LIN {X 0,Y 394.469,Z 685.03,A -85,B 0,C 180,E1 10622.196,E2 10622.196} C_VEL
LIN {X 0,Y 393.966,Z 685.03,A -85,B 0,C 180,E1 10628.817,E2 10628.817} C_VEL
LIN {X 0,Y 393.674,Z 685.03,A -85,B 0,C 180,E1 10635.567,E2 10635.567} C_VEL
LIN {X 0,Y 393.333,Z 685.03,A -85,B 0,C 180,E1 10642.965,E2 10642.965} C_VEL
LIN {X 0,Y 393.105,Z 685.03,A -85,B 0,C 180,E1 10649.938,E2 10649.938} C_VEL
LIN {X 0,Y 392.893,Z 685.03,A -85,B 0,C 180,E1 10656.24,E2 10656.24} C_VEL
LIN {X 0,Y 392.936,Z 685.03,A -85,B 0,C 180,E1 10662.119,E2 10662.119} C_VEL
LIN {X 0,Y 395.462,Z 690.771,A -85,B 0,C 180,E1 10662.638,E2 10662.638} C_VEL
LIN {X 0,Y 416.78,Z 729.542,A -85,B 0,C 180,E1 10666.332,E2 10666.332} C_VEL
LIN {X 0,Y 428.209,Z 756.474,A -85,B 0,C 180,E1 10668.361,E2 10668.361} C_VEL
LIN {X 0,Y 424.245,Z 796.711,A -85,B 0,C 180,E1 10669.819,E2 10669.819} C_VEL
LIN {X 0,Y 419.16,Z 833.859,A -85,B 0,C 180,E1 10671.939,E2 10671.939} C_VEL
LIN {X 0,Y 413.098,Z 871.588,A -85,B 0,C 180,E1 10675.018,E2 10675.018} C_VEL
LIN {X 0,Y 407.027,Z 907.214,A -85,B 0,C 180,E1 10679.043,E2 10679.043} C_VEL
LIN {X 0,Y 402.042,Z 937.236,A -85,B 0,C 180,E1 10683.592,E2 10683.592} C_VEL
LIN {X 0,Y 398.385,Z 962.296,A -85,B 0,C 180,E1 10688.625,E2 10688.625} C_VEL
LIN {X 0,Y 396.268,Z 980.981,A -85,B 0,C 180,E1 10693.688,E2 10693.688} C_VEL
LIN {X 0,Y 395.371,Z 993.17,A -85,B 0,C 180,E1 10698.288,E2 10698.288} C_VEL
LIN {X 0,Y 392.685,Z 996.516,A -85,B 0,C 180,E1 10700.091,E2 10700.091} C_VEL
LIN {X 0,Y 387.255,Z 999.958,A -85,B 0,C 180,E1 10702.863,E2 10702.863} C_VEL
LIN {X 0,Y 387.166,Z 1000.335,A -85,B 0,C 180,E1 10703.185,E2 10703.185} C_VEL
LIN {X 0,Y 387.072,Z 1004.062,A -85,B 0,C 180,E1 10707.766,E2 10707.766} C_VEL
LIN {X 0,Y 387.105,Z 1004.068,A -85,B 0,C 180,E1 10712.234,E2 10712.234} C_VEL
LIN {X 0,Y 387.212,Z 999.067,A -85,B 0,C 180,E1 10717.839,E2 10717.839} C_VEL
LIN {X 0,Y 387.791,Z 988.198,A -85,B 0,C 180,E1 10723.502,E2 10723.502} C_VEL
LIN {X 0,Y 389.429,Z 970.858,A -85,B 0,C 180,E1 10729.23,E2 10729.23} C_VEL
LIN {X 0,Y 392.649,Z 947.513,A -85,B 0,C 180,E1 10734.704,E2 10734.704} C_VEL
LIN {X 0,Y 397.331,Z 919.555,A -85,B 0,C 180,E1 10739.585,E2 10739.585} C_VEL
LIN {X 0,Y 403.125,Z 887.2,A -85,B 0,C 180,E1 10743.835,E2 10743.835} C_VEL
LIN {X 0,Y 409.473,Z 851.855,A -85,B 0,C 180,E1 10747.269,E2 10747.269} C_VEL
LIN {X 0,Y 415.531,Z 813.064,A -85,B 0,C 180,E1 10749.969,E2 10749.969} C_VEL
LIN {X 0,Y 420.802,Z 771.94,A -85,B 0,C 180,E1 10751.807,E2 10751.807} C_VEL
LIN {X 0,Y 421.503,Z 758.027,A -85,B 0,C 180,E1 10752.3,E2 10752.3} C_VEL
LIN {X 0,Y 406.47,Z 724.052,A -85,B 0,C 180,E1 10755.061,E2 10755.061} C_VEL
LIN {X 0,Y 386.866,Z 689.928,A -85,B 0,C 180,E1 10758.649,E2 10758.649} C_VEL
LIN {X 0,Y 385.156,Z 685.03,A -85,B 0,C 180,E1 10759.111,E2 10759.111} C_VEL
LIN {X 0,Y 385.205,Z 685.03,A -85,B 0,C 180,E1 10765.351,E2 10765.351} C_VEL
LIN {X 0,Y 385.298,Z 685.03,A -85,B 0,C 180,E1 10771.965,E2 10771.965} C_VEL
LIN {X 0,Y 385.532,Z 685.03,A -85,B 0,C 180,E1 10779.371,E2 10779.371} C_VEL
LIN {X 0,Y 385.875,Z 685.03,A -85,B 0,C 180,E1 10786.427,E2 10786.427} C_VEL
LIN {X 0,Y 386.183,Z 685.03,A -85,B 0,C 180,E1 10793.264,E2 10793.264} C_VEL
LIN {X 0,Y 386.519,Z 685.03,A -85,B 0,C 180,E1 10799.996,E2 10799.996} C_VEL
LIN {X 0,Y 386.212,Z 685.03,A -85,B 0,C 180,E1 10806.727,E2 10806.727} C_VEL
LIN {X 0,Y 385.892,Z 685.03,A -85,B 0,C 180,E1 10813.564,E2 10813.564} C_VEL
LIN {X 0,Y 385.559,Z 685.03,A -85,B 0,C 180,E1 10820.618,E2 10820.618} C_VEL
LIN {X 0,Y 385.238,Z 685.03,A -85,B 0,C 180,E1 10828.03,E2 10828.03} C_VEL
LIN {X 0,Y 385.121,Z 685.03,A -85,B 0,C 180,E1 10835.988,E2 10835.988} C_VEL
LIN {X 0,Y 385.051,Z 685.03,A -85,B 0,C 180,E1 10841.875,E2 10841.875} C_VEL
LIN {X 0,Y 385.093,Z 685.261,A -85,B 0,C 180,E1 10847.204,E2 10847.204} C_VEL
LIN {X 0,Y 389.899,Z 695.532,A -85,B 0,C 180,E1 10848.478,E2 10848.478} C_VEL
LIN {X 0,Y 403.522,Z 724.973,A -85,B 0,C 180,E1 10852.426,E2 10852.426} C_VEL
LIN {X 0,Y 413.149,Z 753.666,A -85,B 0,C 180,E1 10856.345,E2 10856.345} C_VEL
LIN {X 0,Y 411.811,Z 765.062,A -85,B 0,C 180,E1 10857.501,E2 10857.501} C_VEL
LIN {X 0,Y 405.854,Z 793.487,A -85,B 0,C 180,E1 10860.821,E2 10860.821} C_VEL
LIN {X 0,Y 399.764,Z 819.011,A -85,B 0,C 180,E1 10864.93,E2 10864.93} C_VEL
LIN {X 0,Y 394.494,Z 840.743,A -85,B 0,C 180,E1 10869.863,E2 10869.863} C_VEL
LIN {X 0,Y 390.94,Z 856.405,A -85,B 0,C 180,E1 10875.016,E2 10875.016} C_VEL
LIN {X 0,Y 389.057,Z 866.332,A -85,B 0,C 180,E1 10879.948,E2 10879.948} C_VEL
LIN {X 0,Y 388.111,Z 872.539,A -85,B 0,C 180,E1 10885.54,E2 10885.54} C_VEL
LIN {X 0,Y 387.923,Z 874.065,A -85,B 0,C 180,E1 10890,E2 10890} C_VEL
LIN {X 0,Y 388.096,Z 872.475,A -85,B 0,C 180,E1 10894.46,E2 10894.46} C_VEL
LIN {X 0,Y 389.066,Z 866.191,A -85,B 0,C 180,E1 10900.051,E2 10900.051} C_VEL
LIN {X 0,Y 391.325,Z 854.489,A -85,B 0,C 180,E1 10905.66,E2 10905.66} C_VEL
LIN {X 0,Y 395.094,Z 837.935,A -85,B 0,C 180,E1 10910.788,E2 10910.788} C_VEL
LIN {X 0,Y 400.386,Z 816.384,A -85,B 0,C 180,E1 10915.461,E2 10915.461} C_VEL
LIN {X 0,Y 406.767,Z 789.56,A -85,B 0,C 180,E1 10919.616,E2 10919.616} C_VEL
LIN {X 0,Y 413.018,Z 758.951,A -85,B 0,C 180,E1 10922.981,E2 10922.981} C_VEL
LIN {X 0,Y 412.872,Z 752.781,A -85,B 0,C 180,E1 10923.689,E2 10923.689} C_VEL
LIN {X 0,Y 402.515,Z 722.507,A -85,B 0,C 180,E1 10927.806,E2 10927.806} C_VEL
LIN {X 0,Y 388.97,Z 693.749,A -85,B 0,C 180,E1 10931.663,E2 10931.663} C_VEL
LIN {X 0,Y 385.136,Z 685.03,A -85,B 0,C 180,E1 10932.792,E2 10932.792} C_VEL
LIN {X 0,Y 385.061,Z 685.03,A -85,B 0,C 180,E1 10938.235,E2 10938.235} C_VEL
LIN {X 0,Y 385.145,Z 685.03,A -85,B 0,C 180,E1 10944.015,E2 10944.015} C_VEL
LIN {X 0,Y 385.28,Z 685.03,A -85,B 0,C 180,E1 10951.973,E2 10951.973} C_VEL
LIN {X 0,Y 385.592,Z 685.03,A -85,B 0,C 180,E1 10959.384,E2 10959.384} C_VEL
LIN {X 0,Y 385.996,Z 685.03,A -85,B 0,C 180,E1 10966.44,E2 10966.44} C_VEL
LIN {X 0,Y 386.217,Z 685.03,A -85,B 0,C 180,E1 10973.273,E2 10973.273} C_VEL
LIN {X 0,Y 386.516,Z 685.03,A -85,B 0,C 180,E1 10980.004,E2 10980.004} C_VEL
LIN {X 0,Y 386.217,Z 685.03,A -85,B 0,C 180,E1 10986.735,E2 10986.735} C_VEL
LIN {X 0,Y 385.841,Z 685.03,A -85,B 0,C 180,E1 10993.575,E2 10993.575} C_VEL
LIN {X 0,Y 385.536,Z 685.03,A -85,B 0,C 180,E1 11000.629,E2 11000.629} C_VEL
LIN {X 0,Y 385.212,Z 685.03,A -85,B 0,C 180,E1 11008.042,E2 11008.042} C_VEL
LIN {X 0,Y 384.994,Z 685.03,A -85,B 0,C 180,E1 11014.604,E2 11014.604} C_VEL
LIN {X 0,Y 385.033,Z 685.03,A -85,B 0,C 180,E1 11020.926,E2 11020.926} C_VEL
LIN {X 0,Y 387.41,Z 690.664,A -85,B 0,C 180,E1 11021.467,E2 11021.467} C_VEL
LIN {X 0,Y 408.33,Z 727.687,A -85,B 0,C 180,E1 11025.27,E2 11025.27} C_VEL
LIN {X 0,Y 421.779,Z 758.874,A -85,B 0,C 180,E1 11027.764,E2 11027.764} C_VEL
LIN {X 0,Y 417.238,Z 800.763,A -85,B 0,C 180,E1 11029.384,E2 11029.384} C_VEL
LIN {X 0,Y 411.514,Z 839.57,A -85,B 0,C 180,E1 11031.771,E2 11031.771} C_VEL
LIN {X 0,Y 405.288,Z 875.621,A -85,B 0,C 180,E1 11034.925,E2 11034.925} C_VEL
LIN {X 0,Y 399.319,Z 908.695,A -85,B 0,C 180,E1 11038.853,E2 11038.853} C_VEL
LIN {X 0,Y 394.332,Z 937.229,A -85,B 0,C 180,E1 11043.338,E2 11043.338} C_VEL
LIN {X 0,Y 390.679,Z 961.297,A -85,B 0,C 180,E1 11048.327,E2 11048.327} C_VEL
LIN {X 0,Y 388.419,Z 980.326,A -85,B 0,C 180,E1 11053.641,E2 11053.641} C_VEL
LIN {X 0,Y 387.495,Z 993.239,A -85,B 0,C 180,E1 11058.772,E2 11058.772} C_VEL
LIN {X 0,Y 387.166,Z 1000.335,A -85,B 0,C 180,E1 11063.185,E2 11063.185} C_VEL
LIN {X 0,Y 384.674,Z 1001.967,A -85,B 0,C 180,E1 11065.075,E2 11065.075} C_VEL
LIN {X 0,Y 379.247,Z 1002.868,A -85,B 0,C 180,E1 11068.28,E2 11068.28} C_VEL
LIN {X 0,Y 379.315,Z 1002.752,A -85,B 0,C 180,E1 11072.28,E2 11072.28} C_VEL
LIN {X 0,Y 379.409,Z 997.703,A -85,B 0,C 180,E1 11078.002,E2 11078.002} C_VEL
LIN {X 0,Y 380,Z 986.746,A -85,B 0,C 180,E1 11083.784,E2 11083.784} C_VEL
LIN {X 0,Y 381.696,Z 969.347,A -85,B 0,C 180,E1 11089.636,E2 11089.636} C_VEL
LIN {X 0,Y 385.128,Z 945.977,A -85,B 0,C 180,E1 11095.22,E2 11095.22} C_VEL
LIN {X 0,Y 390.033,Z 917.967,A -85,B 0,C 180,E1 11100.196,E2 11100.196} C_VEL
LIN {X 0,Y 396.254,Z 885.579,A -85,B 0,C 180,E1 11104.504,E2 11104.504} C_VEL
LIN {X 0,Y 402.935,Z 849.628,A -85,B 0,C 180,E1 11108.033,E2 11108.033} C_VEL
LIN {X 0,Y 409.539,Z 809.766,A -85,B 0,C 180,E1 11110.781,E2 11110.781} C_VEL
LIN {X 0,Y 414.765,Z 770.04,A -85,B 0,C 180,E1 11112.535,E2 11112.535} C_VEL
LIN {X 0,Y 414.943,Z 759.988,A -85,B 0,C 180,E1 11112.95,E2 11112.95} C_VEL
LIN {X 0,Y 401.026,Z 728.07,A -85,B 0,C 180,E1 11115.66,E2 11115.66} C_VEL
LIN {X 0,Y 379.762,Z 690.837,A -85,B 0,C 180,E1 11119.725,E2 11119.725} C_VEL
LIN {X 0,Y 377.221,Z 685.03,A -85,B 0,C 180,E1 11120.447,E2 11120.447} C_VEL
LIN {X 0,Y 377.279,Z 685.03,A -85,B 0,C 180,E1 11127.133,E2 11127.133} C_VEL
LIN {X 0,Y 377.354,Z 685.03,A -85,B 0,C 180,E1 11133.901,E2 11133.901} C_VEL
LIN {X 0,Y 377.696,Z 685.03,A -85,B 0,C 180,E1 11141.357,E2 11141.357} C_VEL
LIN {X 0,Y 378.059,Z 685.03,A -85,B 0,C 180,E1 11148.485,E2 11148.485} C_VEL
LIN {X 0,Y 378.439,Z 685.03,A -85,B 0,C 180,E1 11155.453,E2 11155.453} C_VEL
LIN {X 0,Y 378.641,Z 685.03,A -85,B 0,C 180,E1 11162.279,E2 11162.279} C_VEL
LIN {X 0,Y 378.105,Z 685.03,A -85,B 0,C 180,E1 11169.181,E2 11169.181} C_VEL
LIN {X 0,Y 377.776,Z 685.03,A -85,B 0,C 180,E1 11176.533,E2 11176.533} C_VEL
LIN {X 0,Y 377.495,Z 685.03,A -85,B 0,C 180,E1 11183.555,E2 11183.555} C_VEL
LIN {X 0,Y 377.281,Z 685.03,A -85,B 0,C 180,E1 11188.675,E2 11188.675} C_VEL
LIN {X 0,Y 377.153,Z 685.03,A -85,B 0,C 180,E1 11194.057,E2 11194.057} C_VEL
LIN {X 0,Y 377.086,Z 685.03,A -85,B 0,C 180,E1 11200.507,E2 11200.507} C_VEL
LIN {X 0,Y 377.168,Z 685.245,A -85,B 0,C 180,E1 11205.913,E2 11205.913} C_VEL
LIN {X 0,Y 379.824,Z 690.927,A -85,B 0,C 180,E1 11206.651,E2 11206.651} C_VEL
LIN {X 0,Y 394.62,Z 721.775,A -85,B 0,C 180,E1 11210.957,E2 11210.957} C_VEL
LIN {X 0,Y 404.91,Z 751.043,A -85,B 0,C 180,E1 11215.06,E2 11215.06} C_VEL
LIN {X 0,Y 406.767,Z 759.08,A -85,B 0,C 180,E1 11216.189,E2 11216.189} C_VEL
LIN {X 0,Y 400.403,Z 789.521,A -85,B 0,C 180,E1 11219.543,E2 11219.543} C_VEL
LIN {X 0,Y 393.947,Z 815.666,A -85,B 0,C 180,E1 11223.558,E2 11223.558} C_VEL
LIN {X 0,Y 388.432,Z 837.063,A -85,B 0,C 180,E1 11228.133,E2 11228.133} C_VEL
LIN {X 0,Y 384.108,Z 854.534,A -85,B 0,C 180,E1 11233.452,E2 11233.452} C_VEL
LIN {X 0,Y 381.698,Z 865.796,A -85,B 0,C 180,E1 11238.599,E2 11238.599} C_VEL
LIN {X 0,Y 380.556,Z 872.005,A -85,B 0,C 180,E1 11243.168,E2 11243.168} C_VEL
LIN {X 0,Y 380.244,Z 874.971,A -85,B 0,C 180,E1 11247.726,E2 11247.726} C_VEL
LIN {X 0,Y 380.273,Z 874.927,A -85,B 0,C 180,E1 11252.274,E2 11252.274} C_VEL
LIN {X 0,Y 380.74,Z 870.809,A -85,B 0,C 180,E1 11257.829,E2 11257.829} C_VEL
LIN {X 0,Y 382.541,Z 861.208,A -85,B 0,C 180,E1 11263.691,E2 11263.691} C_VEL
LIN {X 0,Y 386.192,Z 845.737,A -85,B 0,C 180,E1 11269.398,E2 11269.398} C_VEL
LIN {X 0,Y 391.174,Z 826.562,A -85,B 0,C 180,E1 11274.197,E2 11274.197} C_VEL
LIN {X 0,Y 397.318,Z 802.17,A -85,B 0,C 180,E1 11278.574,E2 11278.574} C_VEL
LIN {X 0,Y 403.9,Z 773.338,A -85,B 0,C 180,E1 11282.292,E2 11282.292} C_VEL
LIN {X 0,Y 406.826,Z 758.197,A -85,B 0,C 180,E1 11283.806,E2 11283.806} C_VEL
LIN {X 0,Y 397.562,Z 729.268,A -85,B 0,C 180,E1 11287.904,E2 11287.904} C_VEL
LIN {X 0,Y 384.731,Z 700.515,A -85,B 0,C 180,E1 11291.906,E2 11291.906} C_VEL
LIN {X 0,Y 377.233,Z 685.464,A -85,B 0,C 180,E1 11293.954,E2 11293.954} C_VEL
LIN {X 0,Y 377.109,Z 685.03,A -85,B 0,C 180,E1 11300.2,E2 11300.2} C_VEL
LIN {X 0,Y 377.178,Z 685.03,A -85,B 0,C 180,E1 11307.156,E2 11307.156} C_VEL
LIN {X 0,Y 377.392,Z 685.03,A -85,B 0,C 180,E1 11313.914,E2 11313.914} C_VEL
LIN {X 0,Y 377.621,Z 685.03,A -85,B 0,C 180,E1 11318.928,E2 11318.928} C_VEL
LIN {X 0,Y 378.044,Z 685.03,A -85,B 0,C 180,E1 11326.149,E2 11326.149} C_VEL
LIN {X 0,Y 378.3,Z 685.03,A -85,B 0,C 180,E1 11333.132,E2 11333.132} C_VEL
LIN {X 0,Y 378.614,Z 685.03,A -85,B 0,C 180,E1 11340.004,E2 11340.004} C_VEL
LIN {X 0,Y 378.298,Z 685.03,A -85,B 0,C 180,E1 11346.877,E2 11346.877} C_VEL
LIN {X 0,Y 377.893,Z 685.03,A -85,B 0,C 180,E1 11353.866,E2 11353.866} C_VEL
LIN {X 0,Y 377.564,Z 685.03,A -85,B 0,C 180,E1 11361.085,E2 11361.085} C_VEL
LIN {X 0,Y 377.24,Z 685.03,A -85,B 0,C 180,E1 11368.689,E2 11368.689} C_VEL
LIN {X 0,Y 377.085,Z 685.03,A -85,B 0,C 180,E1 11374.075,E2 11374.075} C_VEL
LIN {X 0,Y 377.052,Z 685.03,A -85,B 0,C 180,E1 11379.679,E2 11379.679} C_VEL
LIN {X 0,Y 379.324,Z 690.563,A -85,B 0,C 180,E1 11380.215,E2 11380.215} C_VEL
LIN {X 0,Y 398.731,Z 723.837,A -85,B 0,C 180,E1 11383.94,E2 11383.94} C_VEL
LIN {X 0,Y 412.774,Z 754.299,A -85,B 0,C 180,E1 11386.602,E2 11386.602} C_VEL
LIN {X 0,Y 415.239,Z 763.368,A -85,B 0,C 180,E1 11387.234,E2 11387.234} C_VEL
LIN {X 0,Y 410.471,Z 802.745,A -85,B 0,C 180,E1 11388.846,E2 11388.846} C_VEL
LIN {X 0,Y 404.664,Z 840.071,A -85,B 0,C 180,E1 11391.221,E2 11391.221} C_VEL
LIN {X 0,Y 398.285,Z 875.04,A -85,B 0,C 180,E1 11394.349,E2 11394.349} C_VEL
LIN {X 0,Y 392.213,Z 906.867,A -85,B 0,C 180,E1 11398.188,E2 11398.188} C_VEL
LIN {X 0,Y 386.774,Z 936.506,A -85,B 0,C 180,E1 11402.938,E2 11402.938} C_VEL
LIN {X 0,Y 382.945,Z 960.212,A -85,B 0,C 180,E1 11407.977,E2 11407.977} C_VEL
LIN {X 0,Y 380.596,Z 979.048,A -85,B 0,C 180,E1 11413.371,E2 11413.371} C_VEL
LIN {X 0,Y 379.671,Z 991.824,A -85,B 0,C 180,E1 11418.538,E2 11418.538} C_VEL
LIN {X 0,Y 379.291,Z 1000.166,A -85,B 0,C 180,E1 11424.052,E2 11424.052} C_VEL
LIN {X 0,Y 379.247,Z 1002.868,A -85,B 0,C 180,E1 11428.28,E2 11428.28} C_VEL
LIN {X 0,Y 376.744,Z 1002.771,A -85,B 0,C 180,E1 11430.227,E2 11430.227} C_VEL
LIN {X 0,Y 371.446,Z 1000.742,A -85,B 0,C 180,E1 11433.492,E2 11433.492} C_VEL
LIN {X 0,Y 371.576,Z 996.334,A -85,B 0,C 180,E1 11438.172,E2 11438.172} C_VEL
LIN {X 0,Y 372.179,Z 985.322,A -85,B 0,C 180,E1 11444.08,E2 11444.08} C_VEL
LIN {X 0,Y 373.835,Z 968.933,A -85,B 0,C 180,E1 11449.759,E2 11449.759} C_VEL
LIN {X 0,Y 377.369,Z 945.917,A -85,B 0,C 180,E1 11455.459,E2 11455.459} C_VEL
LIN {X 0,Y 382.621,Z 917.59,A -85,B 0,C 180,E1 11460.64,E2 11460.64} C_VEL
LIN {X 0,Y 388.909,Z 886.419,A -85,B 0,C 180,E1 11464.911,E2 11464.911} C_VEL
LIN {X 0,Y 395.906,Z 850.845,A -85,B 0,C 180,E1 11468.517,E2 11468.517} C_VEL
LIN {X 0,Y 402.668,Z 812.252,A -85,B 0,C 180,E1 11471.287,E2 11471.287} C_VEL
LIN {X 0,Y 408.421,Z 771.614,A -85,B 0,C 180,E1 11473.173,E2 11473.173} C_VEL
LIN {X 0,Y 408.634,Z 762.648,A -85,B 0,C 180,E1 11473.548,E2 11473.548} C_VEL
LIN {X 0,Y 395.064,Z 731.034,A -85,B 0,C 180,E1 11476.374,E2 11476.374} C_VEL
LIN {X 0,Y 375.274,Z 696.408,A -85,B 0,C 180,E1 11480.291,E2 11480.291} C_VEL
LIN {X 0,Y 369.527,Z 686.724,A -85,B 0,C 180,E1 11481.553,E2 11481.553} C_VEL
LIN {X 0,Y 369.369,Z 685.03,A -85,B 0,C 180,E1 11481.758,E2 11481.758} C_VEL
LIN {X 0,Y 369.344,Z 685.03,A -85,B 0,C 180,E1 11489.09,E2 11489.09} C_VEL
LIN {X 0,Y 369.479,Z 685.03,A -85,B 0,C 180,E1 11495.892,E2 11495.892} C_VEL
LIN {X 0,Y 369.881,Z 685.03,A -85,B 0,C 180,E1 11503.403,E2 11503.403} C_VEL
LIN {X 0,Y 370.175,Z 685.03,A -85,B 0,C 180,E1 11510.612,E2 11510.612} C_VEL
LIN {X 0,Y 370.627,Z 685.03,A -85,B 0,C 180,E1 11517.662,E2 11517.662} C_VEL
LIN {X 0,Y 370.738,Z 685.03,A -85,B 0,C 180,E1 11522.328,E2 11522.328} C_VEL
LIN {X 0,Y 370.175,Z 685.03,A -85,B 0,C 180,E1 11529.379,E2 11529.379} C_VEL
LIN {X 0,Y 369.875,Z 685.03,A -85,B 0,C 180,E1 11536.588,E2 11536.588} C_VEL
LIN {X 0,Y 369.503,Z 685.03,A -85,B 0,C 180,E1 11544.097,E2 11544.097} C_VEL
LIN {X 0,Y 369.216,Z 685.03,A -85,B 0,C 180,E1 11552.086,E2 11552.086} C_VEL
LIN {X 0,Y 369.129,Z 685.03,A -85,B 0,C 180,E1 11559.039,E2 11559.039} C_VEL
LIN {X 0,Y 369.209,Z 685.497,A -85,B 0,C 180,E1 11564.543,E2 11564.543} C_VEL
LIN {X 0,Y 372.121,Z 691.113,A -85,B 0,C 180,E1 11565.366,E2 11565.366} C_VEL
LIN {X 0,Y 386.277,Z 720.075,A -85,B 0,C 180,E1 11569.609,E2 11569.609} C_VEL
LIN {X 0,Y 396.286,Z 747.386,A -85,B 0,C 180,E1 11573.553,E2 11573.553} C_VEL
LIN {X 0,Y 400.075,Z 762.156,A -85,B 0,C 180,E1 11575.716,E2 11575.716} C_VEL
LIN {X 0,Y 393.435,Z 792.215,A -85,B 0,C 180,E1 11579.137,E2 11579.137} C_VEL
LIN {X 0,Y 386.558,Z 818.548,A -85,B 0,C 180,E1 11583.327,E2 11583.327} C_VEL
LIN {X 0,Y 380.71,Z 840.29,A -85,B 0,C 180,E1 11588.186,E2 11588.186} C_VEL
LIN {X 0,Y 376.287,Z 857.424,A -85,B 0,C 180,E1 11593.697,E2 11593.697} C_VEL
LIN {X 0,Y 373.683,Z 868.982,A -85,B 0,C 180,E1 11599.53,E2 11599.53} C_VEL
LIN {X 0,Y 372.57,Z 875.167,A -85,B 0,C 180,E1 11605.354,E2 11605.354} C_VEL
LIN {X 0,Y 372.378,Z 876.682,A -85,B 0,C 180,E1 11610,E2 11610} C_VEL
LIN {X 0,Y 372.555,Z 875.105,A -85,B 0,C 180,E1 11614.646,E2 11614.646} C_VEL
LIN {X 0,Y 373.692,Z 868.845,A -85,B 0,C 180,E1 11620.47,E2 11620.47} C_VEL
LIN {X 0,Y 376.311,Z 857.183,A -85,B 0,C 180,E1 11626.302,E2 11626.302} C_VEL
LIN {X 0,Y 380.604,Z 840.441,A -85,B 0,C 180,E1 11631.683,E2 11631.683} C_VEL
LIN {X 0,Y 386.372,Z 819.153,A -85,B 0,C 180,E1 11636.461,E2 11636.461} C_VEL
LIN {X 0,Y 393.055,Z 793.575,A -85,B 0,C 180,E1 11640.576,E2 11640.576} C_VEL
LIN {X 0,Y 399.728,Z 764.006,A -85,B 0,C 180,E1 11644.009,E2 11644.009} C_VEL
LIN {X 0,Y 399.535,Z 758.733,A -85,B 0,C 180,E1 11644.653,E2 11644.653} C_VEL
LIN {X 0,Y 390.24,Z 729.723,A -85,B 0,C 180,E1 11648.89,E2 11648.89} C_VEL
LIN {X 0,Y 377.665,Z 701.656,A -85,B 0,C 180,E1 11652.962,E2 11652.962} C_VEL
LIN {X 0,Y 369.248,Z 685.771,A -85,B 0,C 180,E1 11655.322,E2 11655.322} C_VEL
LIN {X 0,Y 369.152,Z 685.03,A -85,B 0,C 180,E1 11662.191,E2 11662.191} C_VEL
LIN {X 0,Y 369.286,Z 685.03,A -85,B 0,C 180,E1 11669.105,E2 11669.105} C_VEL
LIN {X 0,Y 369.525,Z 685.03,A -85,B 0,C 180,E1 11675.905,E2 11675.905} C_VEL
LIN {X 0,Y 369.951,Z 685.03,A -85,B 0,C 180,E1 11683.416,E2 11683.416} C_VEL
LIN {X 0,Y 370.22,Z 685.03,A -85,B 0,C 180,E1 11690.622,E2 11690.622} C_VEL
LIN {X 0,Y 370.574,Z 685.03,A -85,B 0,C 180,E1 11697.671,E2 11697.671} C_VEL
LIN {X 0,Y 370.741,Z 685.03,A -85,B 0,C 180,E1 11702.337,E2 11702.337} C_VEL
LIN {X 0,Y 370.166,Z 685.03,A -85,B 0,C 180,E1 11709.388,E2 11709.388} C_VEL
LIN {X 0,Y 369.843,Z 685.03,A -85,B 0,C 180,E1 11716.598,E2 11716.598} C_VEL
LIN {X 0,Y 369.48,Z 685.03,A -85,B 0,C 180,E1 11724.108,E2 11724.108} C_VEL
LIN {X 0,Y 369.183,Z 685.03,A -85,B 0,C 180,E1 11732.1,E2 11732.1} C_VEL
LIN {X 0,Y 369.209,Z 685.797,A -85,B 0,C 180,E1 11738.383,E2 11738.383} C_VEL
LIN {X 0,Y 372.149,Z 691.184,A -85,B 0,C 180,E1 11739.052,E2 11739.052} C_VEL
LIN {X 0,Y 393.178,Z 727.529,A -85,B 0,C 180,E1 11743.281,E2 11743.281} C_VEL
LIN {X 0,Y 407.033,Z 758.201,A -85,B 0,C 180,E1 11746.075,E2 11746.075} C_VEL
LIN {X 0,Y 408.902,Z 765.346,A -85,B 0,C 180,E1 11746.609,E2 11746.609} C_VEL
LIN {X 0,Y 403.633,Z 805.798,A -85,B 0,C 180,E1 11748.352,E2 11748.352} C_VEL
LIN {X 0,Y 397.268,Z 843.984,A -85,B 0,C 180,E1 11750.919,E2 11750.919} C_VEL
LIN {X 0,Y 390.172,Z 880.568,A -85,B 0,C 180,E1 11754.411,E2 11754.411} C_VEL
LIN {X 0,Y 383.607,Z 913.124,A -85,B 0,C 180,E1 11758.672,E2 11758.672} C_VEL
LIN {X 0,Y 378.207,Z 941.266,A -85,B 0,C 180,E1 11763.587,E2 11763.587} C_VEL
LIN {X 0,Y 374.426,Z 964.617,A -85,B 0,C 180,E1 11769.042,E2 11769.042} C_VEL
LIN {X 0,Y 372.392,Z 982.303,A -85,B 0,C 180,E1 11774.729,E2 11774.729} C_VEL
LIN {X 0,Y 371.784,Z 992.626,A -85,B 0,C 180,E1 11779.476,E2 11779.476} C_VEL
LIN {X 0,Y 371.486,Z 998.825,A -85,B 0,C 180,E1 11783.927,E2 11783.927} C_VEL
LIN {X 0,Y 371.449,Z 1001.559,A -85,B 0,C 180,E1 11788.282,E2 11788.282} C_VEL
LIN {X 0,Y 371.446,Z 1000.742,A -85,B 0,C 180,E1 11793.492,E2 11793.492} C_VEL
LIN {X 0,Y 368.993,Z 998.993,A -85,B 0,C 180,E1 11795.468,E2 11795.468} C_VEL
LIN {X 0,Y 363.743,Z 994.382,A -85,B 0,C 180,E1 11798.75,E2 11798.75} C_VEL
LIN {X 0,Y 364.342,Z 983.917,A -85,B 0,C 180,E1 11804.389,E2 11804.389} C_VEL
LIN {X 0,Y 366.151,Z 967.494,A -85,B 0,C 180,E1 11810.191,E2 11810.191} C_VEL
LIN {X 0,Y 369.971,Z 944.03,A -85,B 0,C 180,E1 11816.093,E2 11816.093} C_VEL
LIN {X 0,Y 375.525,Z 915.942,A -85,B 0,C 180,E1 11821.304,E2 11821.304} C_VEL
LIN {X 0,Y 382.321,Z 883.591,A -85,B 0,C 180,E1 11825.777,E2 11825.777} C_VEL
LIN {X 0,Y 389.612,Z 848.414,A -85,B 0,C 180,E1 11829.341,E2 11829.341} C_VEL
LIN {X 0,Y 396.757,Z 809.229,A -85,B 0,C 180,E1 11832.14,E2 11832.14} C_VEL
LIN {X 0,Y 402.684,Z 768.292,A -85,B 0,C 180,E1 11833.992,E2 11833.992} C_VEL
LIN {X 0,Y 395.783,Z 748.139,A -85,B 0,C 180,E1 11835.716,E2 11835.716} C_VEL
LIN {X 0,Y 377.634,Z 713.04,A -85,B 0,C 180,E1 11839.432,E2 11839.432} C_VEL
LIN {X 0,Y 363.319,Z 690.196,A -85,B 0,C 180,E1 11842.561,E2 11842.561} C_VEL
LIN {X 0,Y 361.336,Z 685.03,A -85,B 0,C 180,E1 11843.194,E2 11843.194} C_VEL
LIN {X 0,Y 361.414,Z 685.03,A -85,B 0,C 180,E1 11849.929,E2 11849.929} C_VEL
LIN {X 0,Y 361.638,Z 685.03,A -85,B 0,C 180,E1 11857.939,E2 11857.939} C_VEL
LIN {X 0,Y 362.04,Z 685.03,A -85,B 0,C 180,E1 11865.514,E2 11865.514} C_VEL
LIN {X 0,Y 362.428,Z 685.03,A -85,B 0,C 180,E1 11872.821,E2 11872.821} C_VEL
LIN {X 0,Y 362.839,Z 685.03,A -85,B 0,C 180,E1 11879.995,E2 11879.995} C_VEL
LIN {X 0,Y 362.444,Z 685.03,A -85,B 0,C 180,E1 11887.17,E2 11887.17} C_VEL
LIN {X 0,Y 362.046,Z 685.03,A -85,B 0,C 180,E1 11894.476,E2 11894.476} C_VEL
LIN {X 0,Y 361.665,Z 685.03,A -85,B 0,C 180,E1 11902.049,E2 11902.049} C_VEL
LIN {X 0,Y 361.322,Z 685.03,A -85,B 0,C 180,E1 11910.069,E2 11910.069} C_VEL
LIN {X 0,Y 361.205,Z 685.03,A -85,B 0,C 180,E1 11917.462,E2 11917.462} C_VEL
LIN {X 0,Y 361.238,Z 685.738,A -85,B 0,C 180,E1 11923.082,E2 11923.082} C_VEL
LIN {X 0,Y 364.13,Z 691.139,A -85,B 0,C 180,E1 11923.928,E2 11923.928} C_VEL
LIN {X 0,Y 377.904,Z 718.029,A -85,B 0,C 180,E1 11928.132,E2 11928.132} C_VEL
LIN {X 0,Y 388.658,Z 746.727,A -85,B 0,C 180,E1 11932.427,E2 11932.427} C_VEL
LIN {X 0,Y 393.597,Z 764.245,A -85,B 0,C 180,E1 11935.134,E2 11935.134} C_VEL
LIN {X 0,Y 386.781,Z 793.643,A -85,B 0,C 180,E1 11938.546,E2 11938.546} C_VEL
LIN {X 0,Y 379.617,Z 819.927,A -85,B 0,C 180,E1 11942.798,E2 11942.798} C_VEL
LIN {X 0,Y 373.444,Z 841.654,A -85,B 0,C 180,E1 11947.739,E2 11947.739} C_VEL
LIN {X 0,Y 368.769,Z 858.765,A -85,B 0,C 180,E1 11953.355,E2 11953.355} C_VEL
LIN {X 0,Y 366.019,Z 870.303,A -85,B 0,C 180,E1 11959.308,E2 11959.308} C_VEL
LIN {X 0,Y 364.811,Z 876.479,A -85,B 0,C 180,E1 11965.255,E2 11965.255} C_VEL
LIN {X 0,Y 364.595,Z 877.992,A -85,B 0,C 180,E1 11970,E2 11970} C_VEL
LIN {X 0,Y 364.796,Z 876.418,A -85,B 0,C 180,E1 11974.746,E2 11974.746} C_VEL
LIN {X 0,Y 366.029,Z 870.167,A -85,B 0,C 180,E1 11980.691,E2 11980.691} C_VEL
LIN {X 0,Y 368.813,Z 858.526,A -85,B 0,C 180,E1 11986.643,E2 11986.643} C_VEL
LIN {X 0,Y 373.497,Z 841.311,A -85,B 0,C 180,E1 11992.257,E2 11992.257} C_VEL
LIN {X 0,Y 379.712,Z 819.466,A -85,B 0,C 180,E1 11997.195,E2 11997.195} C_VEL
LIN {X 0,Y 386.895,Z 793.036,A -85,B 0,C 180,E1 12001.444,E2 12001.444} C_VEL
LIN {X 0,Y 393.324,Z 763.257,A -85,B 0,C 180,E1 12004.918,E2 12004.918} C_VEL
LIN {X 0,Y 384.479,Z 734.278,A -85,B 0,C 180,E1 12009.316,E2 12009.316} C_VEL
LIN {X 0,Y 373.198,Z 707.77,A -85,B 0,C 180,E1 12013.308,E2 12013.308} C_VEL
LIN {X 0,Y 361.342,Z 686.287,A -85,B 0,C 180,E1 12016.756,E2 12016.756} C_VEL
LIN {X 0,Y 361.249,Z 685.03,A -85,B 0,C 180,E1 12016.917,E2 12016.917} C_VEL
LIN {X 0,Y 361.202,Z 685.03,A -85,B 0,C 180,E1 12024.214,E2 12024.214} C_VEL
LIN {X 0,Y 361.37,Z 685.03,A -85,B 0,C 180,E1 12031.272,E2 12031.272} C_VEL
LIN {X 0,Y 361.69,Z 685.03,A -85,B 0,C 180,E1 12037.952,E2 12037.952} C_VEL
LIN {X 0,Y 362.154,Z 685.03,A -85,B 0,C 180,E1 12045.528,E2 12045.528} C_VEL
LIN {X 0,Y 362.455,Z 685.03,A -85,B 0,C 180,E1 12052.83,E2 12052.83} C_VEL
LIN {X 0,Y 362.834,Z 685.03,A -85,B 0,C 180,E1 12060.005,E2 12060.005} C_VEL
LIN {X 0,Y 362.447,Z 685.03,A -85,B 0,C 180,E1 12067.179,E2 12067.179} C_VEL
LIN {X 0,Y 362.006,Z 685.03,A -85,B 0,C 180,E1 12074.487,E2 12074.487} C_VEL
LIN {X 0,Y 361.643,Z 685.03,A -85,B 0,C 180,E1 12082.061,E2 12082.061} C_VEL
LIN {X 0,Y 361.294,Z 685.03,A -85,B 0,C 180,E1 12088.706,E2 12088.706} C_VEL
LIN {X 0,Y 361.121,Z 685.03,A -85,B 0,C 180,E1 12095.806,E2 12095.806} C_VEL
LIN {X 0,Y 361.155,Z 685.03,A -85,B 0,C 180,E1 12096.884,E2 12096.884} C_VEL
LIN {X 0,Y 363.332,Z 690.428,A -85,B 0,C 180,E1 12097.471,E2 12097.471} C_VEL
LIN {X 0,Y 381.19,Z 719.299,A -85,B 0,C 180,E1 12101.315,E2 12101.315} C_VEL
LIN {X 0,Y 398.135,Z 753.676,A -85,B 0,C 180,E1 12104.81,E2 12104.81} C_VEL
LIN {X 0,Y 402.515,Z 768.228,A -85,B 0,C 180,E1 12105.992,E2 12105.992} C_VEL
LIN {X 0,Y 396.477,Z 810.535,A -85,B 0,C 180,E1 12107.94,E2 12107.94} C_VEL
LIN {X 0,Y 389.535,Z 848.953,A -85,B 0,C 180,E1 12110.714,E2 12110.714} C_VEL
LIN {X 0,Y 382.396,Z 883.575,A -85,B 0,C 180,E1 12114.231,E2 12114.231} C_VEL
LIN {X 0,Y 375.815,Z 914.882,A -85,B 0,C 180,E1 12118.535,E2 12118.535} C_VEL
LIN {X 0,Y 370.453,Z 941.509,A -85,B 0,C 180,E1 12123.38,E2 12123.38} C_VEL
LIN {X 0,Y 366.61,Z 964.252,A -85,B 0,C 180,E1 12128.89,E2 12128.89} C_VEL
LIN {X 0,Y 364.595,Z 980.893,A -85,B 0,C 180,E1 12134.394,E2 12134.394} C_VEL
LIN {X 0,Y 363.97,Z 991.255,A -85,B 0,C 180,E1 12139.248,E2 12139.248} C_VEL
LIN {X 0,Y 363.675,Z 998.319,A -85,B 0,C 180,E1 12144.77,E2 12144.77} C_VEL
LIN {X 0,Y 363.787,Z 1000.617,A -85,B 0,C 180,E1 12150,E2 12150} C_VEL
LIN {X 0,Y 363.713,Z 998.273,A -85,B 0,C 180,E1 12155.296,E2 12155.296} C_VEL
LIN {X 0,Y 363.743,Z 994.382,A -85,B 0,C 180,E1 12158.75,E2 12158.75} C_VEL
LIN {X 0,Y 361.402,Z 991.009,A -85,B 0,C 180,E1 12160.719,E2 12160.719} C_VEL
LIN {X 0,Y 356.426,Z 984.095,A -85,B 0,C 180,E1 12163.979,E2 12163.979} C_VEL
LIN {X 0,Y 358.016,Z 968.992,A -85,B 0,C 180,E1 12169.706,E2 12169.706} C_VEL
LIN {X 0,Y 361.476,Z 947.906,A -85,B 0,C 180,E1 12175.45,E2 12175.45} C_VEL
LIN {X 0,Y 366.828,Z 921.728,A -85,B 0,C 180,E1 12180.744,E2 12180.744} C_VEL
LIN {X 0,Y 373.941,Z 889.663,A -85,B 0,C 180,E1 12185.574,E2 12185.574} C_VEL
LIN {X 0,Y 381.895,Z 853.551,A -85,B 0,C 180,E1 12189.517,E2 12189.517} C_VEL
LIN {X 0,Y 389.188,Z 816.502,A -85,B 0,C 180,E1 12192.377,E2 12192.377} C_VEL
LIN {X 0,Y 395.369,Z 777.872,A -85,B 0,C 180,E1 12194.362,E2 12194.362} C_VEL
LIN {X 0,Y 396.028,Z 767.634,A -85,B 0,C 180,E1 12194.835,E2 12194.835} C_VEL
LIN {X 0,Y 383.152,Z 736.972,A -85,B 0,C 180,E1 12197.873,E2 12197.873} C_VEL
LIN {X 0,Y 363.95,Z 702.946,A -85,B 0,C 180,E1 12202.049,E2 12202.049} C_VEL
LIN {X 0,Y 353.499,Z 686.261,A -85,B 0,C 180,E1 12204.59,E2 12204.59} C_VEL
LIN {X 0,Y 353.4,Z 685.03,A -85,B 0,C 180,E1 12204.673,E2 12204.673} C_VEL
LIN {X 0,Y 353.478,Z 685.03,A -85,B 0,C 180,E1 12211.989,E2 12211.989} C_VEL
LIN {X 0,Y 353.797,Z 685.03,A -85,B 0,C 180,E1 12220.046,E2 12220.046} C_VEL
LIN {X 0,Y 354.253,Z 685.03,A -85,B 0,C 180,E1 12227.699,E2 12227.699} C_VEL
LIN {X 0,Y 354.673,Z 685.03,A -85,B 0,C 180,E1 12235.114,E2 12235.114} C_VEL
LIN {X 0,Y 354.926,Z 685.03,A -85,B 0,C 180,E1 12242.432,E2 12242.432} C_VEL
LIN {X 0,Y 354.318,Z 685.03,A -85,B 0,C 180,E1 12249.803,E2 12249.803} C_VEL
LIN {X 0,Y 353.967,Z 685.03,A -85,B 0,C 180,E1 12257.356,E2 12257.356} C_VEL
LIN {X 0,Y 353.561,Z 685.03,A -85,B 0,C 180,E1 12265.257,E2 12265.257} C_VEL
LIN {X 0,Y 353.294,Z 685.03,A -85,B 0,C 180,E1 12271.324,E2 12271.324} C_VEL
LIN {X 0,Y 353.26,Z 685.03,A -85,B 0,C 180,E1 12276.72,E2 12276.72} C_VEL
LIN {X 0,Y 353.342,Z 685.649,A -85,B 0,C 180,E1 12281.506,E2 12281.506} C_VEL
LIN {X 0,Y 355.888,Z 690.848,A -85,B 0,C 180,E1 12282.309,E2 12282.309} C_VEL
LIN {X 0,Y 369.227,Z 715.718,A -85,B 0,C 180,E1 12286.511,E2 12286.511} C_VEL
LIN {X 0,Y 379.91,Z 742.464,A -85,B 0,C 180,E1 12290.71,E2 12290.71} C_VEL
LIN {X 0,Y 386.976,Z 767.157,A -85,B 0,C 180,E1 12294.622,E2 12294.622} C_VEL
LIN {X 0,Y 379.615,Z 797.045,A -85,B 0,C 180,E1 12298.218,E2 12298.218} C_VEL
LIN {X 0,Y 372.261,Z 822.794,A -85,B 0,C 180,E1 12302.542,E2 12302.542} C_VEL
LIN {X 0,Y 365.904,Z 844.111,A -85,B 0,C 180,E1 12307.575,E2 12307.575} C_VEL
LIN {X 0,Y 361.281,Z 860.1,A -85,B 0,C 180,E1 12313,E2 12313} C_VEL
LIN {X 0,Y 358.349,Z 871.624,A -85,B 0,C 180,E1 12319.077,E2 12319.077} C_VEL
LIN {X 0,Y 357.036,Z 877.794,A -85,B 0,C 180,E1 12325.151,E2 12325.151} C_VEL
LIN {X 0,Y 356.805,Z 879.304,A -85,B 0,C 180,E1 12330,E2 12330} C_VEL
LIN {X 0,Y 357.022,Z 877.733,A -85,B 0,C 180,E1 12334.849,E2 12334.849} C_VEL
LIN {X 0,Y 358.361,Z 871.489,A -85,B 0,C 180,E1 12340.923,E2 12340.923} C_VEL
LIN {X 0,Y 361.326,Z 859.867,A -85,B 0,C 180,E1 12346.998,E2 12346.998} C_VEL
LIN {X 0,Y 366.272,Z 842.673,A -85,B 0,C 180,E1 12352.721,E2 12352.721} C_VEL
LIN {X 0,Y 372.792,Z 820.854,A -85,B 0,C 180,E1 12357.742,E2 12357.742} C_VEL
LIN {X 0,Y 380.29,Z 794.467,A -85,B 0,C 180,E1 12362.054,E2 12362.054} C_VEL
LIN {X 0,Y 386.748,Z 766.298,A -85,B 0,C 180,E1 12365.422,E2 12365.422} C_VEL
LIN {X 0,Y 378.368,Z 737.837,A -85,B 0,C 180,E1 12369.905,E2 12369.905} C_VEL
LIN {X 0,Y 366.425,Z 709.767,A -85,B 0,C 180,E1 12374.336,E2 12374.336} C_VEL
LIN {X 0,Y 354.89,Z 689.742,A -85,B 0,C 180,E1 12377.841,E2 12377.841} C_VEL
LIN {X 0,Y 353.332,Z 685.03,A -85,B 0,C 180,E1 12378.491,E2 12378.491} C_VEL
LIN {X 0,Y 353.299,Z 685.03,A -85,B 0,C 180,E1 12386.281,E2 12386.281} C_VEL
LIN {X 0,Y 353.501,Z 685.03,A -85,B 0,C 180,E1 12393.692,E2 12393.692} C_VEL
LIN {X 0,Y 353.861,Z 685.03,A -85,B 0,C 180,E1 12400.06,E2 12400.06} C_VEL
LIN {X 0,Y 354.349,Z 685.03,A -85,B 0,C 180,E1 12407.712,E2 12407.712} C_VEL
LIN {X 0,Y 354.672,Z 685.03,A -85,B 0,C 180,E1 12415.124,E2 12415.124} C_VEL
LIN {X 0,Y 354.928,Z 685.03,A -85,B 0,C 180,E1 12422.441,E2 12422.441} C_VEL
LIN {X 0,Y 354.3,Z 685.03,A -85,B 0,C 180,E1 12429.813,E2 12429.813} C_VEL
LIN {X 0,Y 353.918,Z 685.03,A -85,B 0,C 180,E1 12437.369,E2 12437.369} C_VEL
LIN {X 0,Y 353.538,Z 685.03,A -85,B 0,C 180,E1 12445.27,E2 12445.27} C_VEL
LIN {X 0,Y 353.256,Z 685.03,A -85,B 0,C 180,E1 12451.314,E2 12451.314} C_VEL
LIN {X 0,Y 353.206,Z 685.441,A -85,B 0,C 180,E1 12455.347,E2 12455.347} C_VEL
LIN {X 0,Y 355.722,Z 690.756,A -85,B 0,C 180,E1 12456.03,E2 12456.03} C_VEL
LIN {X 0,Y 374.218,Z 720.361,A -85,B 0,C 180,E1 12460.247,E2 12460.247} C_VEL
LIN {X 0,Y 391.036,Z 754.162,A -85,B 0,C 180,E1 12463.902,E2 12463.902} C_VEL
LIN {X 0,Y 396.334,Z 769.692,A -85,B 0,C 180,E1 12465.312,E2 12465.312} C_VEL
LIN {X 0,Y 390.208,Z 810.157,A -85,B 0,C 180,E1 12467.228,E2 12467.228} C_VEL
LIN {X 0,Y 383.129,Z 847.699,A -85,B 0,C 180,E1 12469.972,E2 12469.972} C_VEL
LIN {X 0,Y 375.854,Z 881.362,A -85,B 0,C 180,E1 12473.416,E2 12473.416} C_VEL
LIN {X 0,Y 368.694,Z 913.343,A -85,B 0,C 180,E1 12477.855,E2 12477.855} C_VEL
LIN {X 0,Y 362.987,Z 940.01,A -85,B 0,C 180,E1 12482.788,E2 12482.788} C_VEL
LIN {X 0,Y 358.944,Z 962.805,A -85,B 0,C 180,E1 12488.417,E2 12488.417} C_VEL
LIN {X 0,Y 356.806,Z 979.493,A -85,B 0,C 180,E1 12494.044,E2 12494.044} C_VEL
LIN {X 0,Y 356.136,Z 989.888,A -85,B 0,C 180,E1 12499.008,E2 12499.008} C_VEL
LIN {X 0,Y 355.856,Z 996.379,A -85,B 0,C 180,E1 12503.915,E2 12503.915} C_VEL
LIN {X 0,Y 356,Z 999.306,A -85,B 0,C 180,E1 12510,E2 12510} C_VEL
LIN {X 0,Y 355.928,Z 997.398,A -85,B 0,C 180,E1 12514.864,E2 12514.864} C_VEL
LIN {X 0,Y 355.989,Z 991.839,A -85,B 0,C 180,E1 12519.762,E2 12519.762} C_VEL
LIN {X 0,Y 356.426,Z 984.095,A -85,B 0,C 180,E1 12523.979,E2 12523.979} C_VEL
LIN {X 0,Y 353.047,Z 977.771,A -85,B 0,C 180,E1 12526.562,E2 12526.562} C_VEL
LIN {X 0,Y 349.903,Z 970.652,A -85,B 0,C 180,E1 12529.145,E2 12529.145} C_VEL
LIN {X 0,Y 353.41,Z 949.565,A -85,B 0,C 180,E1 12535.276,E2 12535.276} C_VEL
LIN {X 0,Y 359.099,Z 922.895,A -85,B 0,C 180,E1 12540.94,E2 12540.94} C_VEL
LIN {X 0,Y 366.198,Z 892.165,A -85,B 0,C 180,E1 12545.785,E2 12545.785} C_VEL
LIN {X 0,Y 374.327,Z 857.442,A -85,B 0,C 180,E1 12549.788,E2 12549.788} C_VEL
LIN {X 0,Y 382.44,Z 818.807,A -85,B 0,C 180,E1 12552.941,E2 12552.941} C_VEL
LIN {X 0,Y 389.227,Z 778.674,A -85,B 0,C 180,E1 12555.079,E2 12555.079} C_VEL
LIN {X 0,Y 389.683,Z 769.915,A -85,B 0,C 180,E1 12555.519,E2 12555.519} C_VEL
LIN {X 0,Y 377.152,Z 739.68,A -85,B 0,C 180,E1 12558.685,E2 12558.685} C_VEL
LIN {X 0,Y 359.316,Z 708.004,A -85,B 0,C 180,E1 12562.744,E2 12562.744} C_VEL
LIN {X 0,Y 347.986,Z 690.799,A -85,B 0,C 180,E1 12565.589,E2 12565.589} C_VEL
LIN {X 0,Y 345.496,Z 685.03,A -85,B 0,C 180,E1 12566.452,E2 12566.452} C_VEL
LIN {X 0,Y 345.622,Z 685.03,A -85,B 0,C 180,E1 12574.109,E2 12574.109} C_VEL
LIN {X 0,Y 345.992,Z 685.03,A -85,B 0,C 180,E1 12582.22,E2 12582.22} C_VEL
LIN {X 0,Y 346.393,Z 685.03,A -85,B 0,C 180,E1 12589.961,E2 12589.961} C_VEL
LIN {X 0,Y 346.941,Z 685.03,A -85,B 0,C 180,E1 12597.503,E2 12597.503} C_VEL
LIN {X 0,Y 347.031,Z 685.03,A -85,B 0,C 180,E1 12602.487,E2 12602.487} C_VEL
LIN {X 0,Y 346.392,Z 685.03,A -85,B 0,C 180,E1 12610.03,E2 12610.03} C_VEL
LIN {X 0,Y 345.995,Z 685.03,A -85,B 0,C 180,E1 12617.769,E2 12617.769} C_VEL
LIN {X 0,Y 345.621,Z 685.03,A -85,B 0,C 180,E1 12625.88,E2 12625.88} C_VEL
LIN {X 0,Y 345.363,Z 685.03,A -85,B 0,C 180,E1 12633.884,E2 12633.884} C_VEL
LIN {X 0,Y 345.394,Z 685.649,A -85,B 0,C 180,E1 12639.789,E2 12639.789} C_VEL
LIN {X 0,Y 348.195,Z 691.049,A -85,B 0,C 180,E1 12640.703,E2 12640.703} C_VEL
LIN {X 0,Y 361.699,Z 715.652,A -85,B 0,C 180,E1 12645.162,E2 12645.162} C_VEL
LIN {X 0,Y 372.738,Z 742.81,A -85,B 0,C 180,E1 12649.628,E2 12649.628} C_VEL
LIN {X 0,Y 380.321,Z 770.069,A -85,B 0,C 180,E1 12654.095,E2 12654.095} C_VEL
LIN {X 0,Y 373.029,Z 798.464,A -85,B 0,C 180,E1 12657.589,E2 12657.589} C_VEL
LIN {X 0,Y 365.373,Z 824.171,A -85,B 0,C 180,E1 12661.979,E2 12661.979} C_VEL
LIN {X 0,Y 358.688,Z 845.467,A -85,B 0,C 180,E1 12667.099,E2 12667.099} C_VEL
LIN {X 0,Y 353.79,Z 861.436,A -85,B 0,C 180,E1 12672.629,E2 12672.629} C_VEL
LIN {X 0,Y 350.675,Z 872.946,A -85,B 0,C 180,E1 12678.835,E2 12678.835} C_VEL
LIN {X 0,Y 349.279,Z 879.105,A -85,B 0,C 180,E1 12685.043,E2 12685.043} C_VEL
LIN {X 0,Y 349.022,Z 880.614,A -85,B 0,C 180,E1 12690,E2 12690} C_VEL
LIN {X 0,Y 349.265,Z 879.046,A -85,B 0,C 180,E1 12694.957,E2 12694.957} C_VEL
LIN {X 0,Y 350.688,Z 872.813,A -85,B 0,C 180,E1 12701.165,E2 12701.165} C_VEL
LIN {X 0,Y 353.855,Z 861.205,A -85,B 0,C 180,E1 12707.368,E2 12707.368} C_VEL
LIN {X 0,Y 359.079,Z 844.031,A -85,B 0,C 180,E1 12713.202,E2 12713.202} C_VEL
LIN {X 0,Y 365.924,Z 822.235,A -85,B 0,C 180,E1 12718.31,E2 12718.31} C_VEL
LIN {X 0,Y 373.73,Z 795.892,A -85,B 0,C 180,E1 12722.686,E2 12722.686} C_VEL
LIN {X 0,Y 380.015,Z 768.888,A -85,B 0,C 180,E1 12726.01,E2 12726.01} C_VEL
LIN {X 0,Y 372.04,Z 740.86,A -85,B 0,C 180,E1 12730.59,E2 12730.59} C_VEL
LIN {X 0,Y 361.002,Z 713.903,A -85,B 0,C 180,E1 12734.995,E2 12734.995} C_VEL
LIN {X 0,Y 347.682,Z 690.563,A -85,B 0,C 180,E1 12739.318,E2 12739.318} C_VEL
LIN {X 0,Y 345.393,Z 685.03,A -85,B 0,C 180,E1 12740.21,E2 12740.21} C_VEL
LIN {X 0,Y 345.419,Z 685.03,A -85,B 0,C 180,E1 12748.392,E2 12748.392} C_VEL
LIN {X 0,Y 345.72,Z 685.03,A -85,B 0,C 180,E1 12756.434,E2 12756.434} C_VEL
LIN {X 0,Y 346.137,Z 685.03,A -85,B 0,C 180,E1 12763.556,E2 12763.556} C_VEL
LIN {X 0,Y 346.443,Z 685.03,A -85,B 0,C 180,E1 12769.972,E2 12769.972} C_VEL
LIN {X 0,Y 346.888,Z 685.03,A -85,B 0,C 180,E1 12777.512,E2 12777.512} C_VEL
LIN {X 0,Y 347.034,Z 685.03,A -85,B 0,C 180,E1 12782.497,E2 12782.497} C_VEL
LIN {X 0,Y 346.37,Z 685.03,A -85,B 0,C 180,E1 12790.04,E2 12790.04} C_VEL
LIN {X 0,Y 345.954,Z 685.03,A -85,B 0,C 180,E1 12797.782,E2 12797.782} C_VEL
LIN {X 0,Y 345.596,Z 685.03,A -85,B 0,C 180,E1 12805.893,E2 12805.893} C_VEL
LIN {X 0,Y 345.309,Z 685.03,A -85,B 0,C 180,E1 12813.645,E2 12813.645} C_VEL
LIN {X 0,Y 347.621,Z 690.651,A -85,B 0,C 180,E1 12814.358,E2 12814.358} C_VEL
LIN {X 0,Y 363.495,Z 714.916,A -85,B 0,C 180,E1 12818.261,E2 12818.261} C_VEL
LIN {X 0,Y 380.954,Z 747.745,A -85,B 0,C 180,E1 12822.235,E2 12822.235} C_VEL
LIN {X 0,Y 390.027,Z 771.956,A -85,B 0,C 180,E1 12824.651,E2 12824.651} C_VEL
LIN {X 0,Y 383.89,Z 810.339,A -85,B 0,C 180,E1 12826.525,E2 12826.525} C_VEL
LIN {X 0,Y 376.404,Z 848.099,A -85,B 0,C 180,E1 12829.35,E2 12829.35} C_VEL
LIN {X 0,Y 368.913,Z 881.13,A -85,B 0,C 180,E1 12832.813,E2 12832.813} C_VEL
LIN {X 0,Y 361.69,Z 911.827,A -85,B 0,C 180,E1 12837.155,E2 12837.155} C_VEL
LIN {X 0,Y 355.301,Z 940.012,A -85,B 0,C 180,E1 12842.498,E2 12842.498} C_VEL
LIN {X 0,Y 351.127,Z 962.455,A -85,B 0,C 180,E1 12848.243,E2 12848.243} C_VEL
LIN {X 0,Y 348.865,Z 979.617,A -85,B 0,C 180,E1 12854.316,E2 12854.316} C_VEL
LIN {X 0,Y 348.216,Z 990.495,A -85,B 0,C 180,E1 12860.018,E2 12860.018} C_VEL
LIN {X 0,Y 348.03,Z 996.609,A -85,B 0,C 180,E1 12865.746,E2 12865.746} C_VEL
LIN {X 0,Y 348.215,Z 997.995,A -85,B 0,C 180,E1 12870,E2 12870} C_VEL
LIN {X 0,Y 348.11,Z 996.073,A -85,B 0,C 180,E1 12874.974,E2 12874.974} C_VEL
LIN {X 0,Y 348.178,Z 990.492,A -85,B 0,C 180,E1 12879.983,E2 12879.983} C_VEL
LIN {X 0,Y 348.88,Z 979.623,A -85,B 0,C 180,E1 12885.684,E2 12885.684} C_VEL
LIN {X 0,Y 349.903,Z 970.652,A -85,B 0,C 180,E1 12889.145,E2 12889.145} C_VEL
LIN {X 0,Y 347.033,Z 962.97,A -85,B 0,C 180,E1 12891.699,E2 12891.699} C_VEL
LIN {X 0,Y 344.726,Z 954.335,A -85,B 0,C 180,E1 12894.209,E2 12894.209} C_VEL
LIN {X 0,Y 350.048,Z 929.324,A -85,B 0,C 180,E1 12900.103,E2 12900.103} C_VEL
LIN {X 0,Y 357.377,Z 899.463,A -85,B 0,C 180,E1 12905.291,E2 12905.291} C_VEL
LIN {X 0,Y 365.576,Z 866.307,A -85,B 0,C 180,E1 12909.527,E2 12909.527} C_VEL
LIN {X 0,Y 373.997,Z 829.35,A -85,B 0,C 180,E1 12912.911,E2 12912.911} C_VEL
LIN {X 0,Y 381.413,Z 790.164,A -85,B 0,C 180,E1 12915.328,E2 12915.328} C_VEL
LIN {X 0,Y 383.475,Z 772.778,A -85,B 0,C 180,E1 12916.167,E2 12916.167} C_VEL
LIN {X 0,Y 371.866,Z 743.964,A -85,B 0,C 180,E1 12919.32,E2 12919.32} C_VEL
LIN {X 0,Y 354.783,Z 712.959,A -85,B 0,C 180,E1 12923.452,E2 12923.452} C_VEL
LIN {X 0,Y 340.151,Z 690.882,A -85,B 0,C 180,E1 12927.342,E2 12927.342} C_VEL
LIN {X 0,Y 337.612,Z 685.701,A -85,B 0,C 180,E1 12928.143,E2 12928.143} C_VEL
LIN {X 0,Y 337.775,Z 685.03,A -85,B 0,C 180,E1 12936.289,E2 12936.289} C_VEL
LIN {X 0,Y 338.016,Z 685.03,A -85,B 0,C 180,E1 12941.786,E2 12941.786} C_VEL
LIN {X 0,Y 338.455,Z 685.03,A -85,B 0,C 180,E1 12949.723,E2 12949.723} C_VEL
LIN {X 0,Y 339.026,Z 685.03,A -85,B 0,C 180,E1 12957.444,E2 12957.444} C_VEL
LIN {X 0,Y 339.112,Z 685.03,A -85,B 0,C 180,E1 12962.545,E2 12962.545} C_VEL
LIN {X 0,Y 338.453,Z 685.03,A -85,B 0,C 180,E1 12970.267,E2 12970.267} C_VEL
LIN {X 0,Y 338.022,Z 685.03,A -85,B 0,C 180,E1 12978.203,E2 12978.203} C_VEL
LIN {X 0,Y 337.788,Z 685.03,A -85,B 0,C 180,E1 12983.7,E2 12983.7} C_VEL
LIN {X 0,Y 337.467,Z 685.03,A -85,B 0,C 180,E1 12991.833,E2 12991.833} C_VEL
LIN {X 0,Y 337.376,Z 685.471,A -85,B 0,C 180,E1 12997.887,E2 12997.887} C_VEL
LIN {X 0,Y 339.975,Z 690.899,A -85,B 0,C 180,E1 12998.817,E2 12998.817} C_VEL
LIN {X 0,Y 351.774,Z 710.862,A -85,B 0,C 180,E1 13002.832,E2 13002.832} C_VEL
LIN {X 0,Y 363.605,Z 737.669,A -85,B 0,C 180,E1 13007.557,E2 13007.557} C_VEL
LIN {X 0,Y 371.539,Z 763.941,A -85,B 0,C 180,E1 13011.976,E2 13011.976} C_VEL
LIN {X 0,Y 373.424,Z 774.179,A -85,B 0,C 180,E1 13013.682,E2 13013.682} C_VEL
LIN {X 0,Y 365.335,Z 803.835,A -85,B 0,C 180,E1 13017.523,E2 13017.523} C_VEL
LIN {X 0,Y 357.098,Z 829.834,A -85,B 0,C 180,E1 13022.301,E2 13022.301} C_VEL
LIN {X 0,Y 350.293,Z 850.38,A -85,B 0,C 180,E1 13027.703,E2 13027.703} C_VEL
LIN {X 0,Y 345.508,Z 865.33,A -85,B 0,C 180,E1 13033.419,E2 13033.419} C_VEL
LIN {X 0,Y 342.621,Z 875.954,A -85,B 0,C 180,E1 13039.853,E2 13039.853} C_VEL
LIN {X 0,Y 341.535,Z 880.415,A -85,B 0,C 180,E1 13044.93,E2 13044.93} C_VEL
LIN {X 0,Y 341.232,Z 881.925,A -85,B 0,C 180,E1 13050,E2 13050} C_VEL
LIN {X 0,Y 341.496,Z 880.36,A -85,B 0,C 180,E1 13055.07,E2 13055.07} C_VEL
LIN {X 0,Y 343.017,Z 874.136,A -85,B 0,C 180,E1 13061.418,E2 13061.418} C_VEL
LIN {X 0,Y 346.378,Z 862.545,A -85,B 0,C 180,E1 13067.755,E2 13067.755} C_VEL
LIN {X 0,Y 351.91,Z 845.386,A -85,B 0,C 180,E1 13073.703,E2 13073.703} C_VEL
LIN {X 0,Y 359.084,Z 823.615,A -85,B 0,C 180,E1 13078.899,E2 13078.899} C_VEL
LIN {X 0,Y 367.211,Z 797.314,A -85,B 0,C 180,E1 13083.341,E2 13083.341} C_VEL
LIN {X 0,Y 373.615,Z 772.807,A -85,B 0,C 180,E1 13086.381,E2 13086.381} C_VEL
LIN {X 0,Y 366.715,Z 746.704,A -85,B 0,C 180,E1 13090.811,E2 13090.811} C_VEL
LIN {X 0,Y 356.386,Z 720.065,A -85,B 0,C 180,E1 13095.358,E2 13095.358} C_VEL
LIN {X 0,Y 343.265,Z 696.291,A -85,B 0,C 180,E1 13099.931,E2 13099.931} C_VEL
LIN {X 0,Y 339.873,Z 690.761,A -85,B 0,C 180,E1 13101.087,E2 13101.087} C_VEL
LIN {X 0,Y 337.401,Z 685.817,A -85,B 0,C 180,E1 13101.957,E2 13101.957} C_VEL
LIN {X 0,Y 337.498,Z 685.03,A -85,B 0,C 180,E1 13108.159,E2 13108.159} C_VEL
LIN {X 0,Y 337.814,Z 685.03,A -85,B 0,C 180,E1 13116.302,E2 13116.302} C_VEL
LIN {X 0,Y 338.092,Z 685.03,A -85,B 0,C 180,E1 13121.801,E2 13121.801} C_VEL
LIN {X 0,Y 338.454,Z 685.03,A -85,B 0,C 180,E1 13128.773,E2 13128.773} C_VEL
LIN {X 0,Y 338.83,Z 685.03,A -85,B 0,C 180,E1 13134.895,E2 13134.895} C_VEL
LIN {X 0,Y 339.115,Z 685.03,A -85,B 0,C 180,E1 13142.555,E2 13142.555} C_VEL
LIN {X 0,Y 338.43,Z 685.03,A -85,B 0,C 180,E1 13150.278,E2 13150.278} C_VEL
LIN {X 0,Y 337.985,Z 685.03,A -85,B 0,C 180,E1 13158.215,E2 13158.215} C_VEL
LIN {X 0,Y 337.77,Z 685.03,A -85,B 0,C 180,E1 13163.712,E2 13163.712} C_VEL
LIN {X 0,Y 337.42,Z 685.03,A -85,B 0,C 180,E1 13171.82,E2 13171.82} C_VEL
LIN {X 0,Y 339.469,Z 690.38,A -85,B 0,C 180,E1 13172.512,E2 13172.512} C_VEL
LIN {X 0,Y 342.266,Z 694.191,A -85,B 0,C 180,E1 13173.299,E2 13173.299} C_VEL
LIN {X 0,Y 357.539,Z 717.825,A -85,B 0,C 180,E1 13177.259,E2 13177.259} C_VEL
LIN {X 0,Y 373.582,Z 747.605,A -85,B 0,C 180,E1 13181.122,E2 13181.122} C_VEL
LIN {X 0,Y 383.804,Z 774.086,A -85,B 0,C 180,E1 13183.964,E2 13183.964} C_VEL
LIN {X 0,Y 377.246,Z 812.546,A -85,B 0,C 180,E1 13185.925,E2 13185.925} C_VEL
LIN {X 0,Y 369.185,Z 850.778,A -85,B 0,C 180,E1 13188.908,E2 13188.908} C_VEL
LIN {X 0,Y 360.617,Z 886.348,A -85,B 0,C 180,E1 13192.866,E2 13192.866} C_VEL
LIN {X 0,Y 352.851,Z 917.688,A -85,B 0,C 180,E1 13197.685,E2 13197.685} C_VEL
LIN {X 0,Y 346.797,Z 944.188,A -85,B 0,C 180,E1 13203.181,E2 13203.181} C_VEL
LIN {X 0,Y 342.662,Z 966.148,A -85,B 0,C 180,E1 13209.372,E2 13209.372} C_VEL
LIN {X 0,Y 340.802,Z 981.099,A -85,B 0,C 180,E1 13215.251,E2 13215.251} C_VEL
LIN {X 0,Y 340.302,Z 990.943,A -85,B 0,C 180,E1 13221.072,E2 13221.072} C_VEL
LIN {X 0,Y 340.303,Z 994.747,A -85,B 0,C 180,E1 13224.912,E2 13224.912} C_VEL
LIN {X 0,Y 340.431,Z 996.685,A -85,B 0,C 180,E1 13230,E2 13230} C_VEL
LIN {X 0,Y 340.316,Z 994.753,A -85,B 0,C 180,E1 13235.088,E2 13235.088} C_VEL
LIN {X 0,Y 340.365,Z 989.145,A -85,B 0,C 180,E1 13240.215,E2 13240.215} C_VEL
LIN {X 0,Y 341.121,Z 978.24,A -85,B 0,C 180,E1 13246.05,E2 13246.05} C_VEL
LIN {X 0,Y 343.569,Z 960.966,A -85,B 0,C 180,E1 13252.285,E2 13252.285} C_VEL
LIN {X 0,Y 344.726,Z 954.335,A -85,B 0,C 180,E1 13254.209,E2 13254.209} C_VEL
LIN {X 0,Y 344.402,Z 949.859,A -85,B 0,C 180,E1 13255.452,E2 13255.452} C_VEL
LIN {X 0,Y 340.775,Z 936.912,A -85,B 0,C 180,E1 13258.832,E2 13258.832} C_VEL
LIN {X 0,Y 341.016,Z 935.61,A -85,B 0,C 180,E1 13259.128,E2 13259.128} C_VEL
LIN {X 0,Y 348.277,Z 906.876,A -85,B 0,C 180,E1 13264.671,E2 13264.671} C_VEL
LIN {X 0,Y 356.943,Z 873.66,A -85,B 0,C 180,E1 13269.355,E2 13269.355} C_VEL
LIN {X 0,Y 365.646,Z 838.314,A -85,B 0,C 180,E1 13272.917,E2 13272.917} C_VEL
LIN {X 0,Y 373.592,Z 799.951,A -85,B 0,C 180,E1 13275.6,E2 13275.6} C_VEL
LIN {X 0,Y 377.284,Z 775.245,A -85,B 0,C 180,E1 13276.866,E2 13276.866} C_VEL
LIN {X 0,Y 365.647,Z 746.159,A -85,B 0,C 180,E1 13280.23,E2 13280.23} C_VEL
LIN {X 0,Y 348.62,Z 715.049,A -85,B 0,C 180,E1 13284.622,E2 13284.622} C_VEL
LIN {X 0,Y 332.784,Z 691.351,A -85,B 0,C 180,E1 13289.126,E2 13289.126} C_VEL
LIN {X 0,Y 329.85,Z 686.931,A -85,B 0,C 180,E1 13290.072,E2 13290.072} C_VEL
LIN {X 0,Y 329.655,Z 685.03,A -85,B 0,C 180,E1 13290.426,E2 13290.426} C_VEL
LIN {X 0,Y 329.897,Z 685.03,A -85,B 0,C 180,E1 13298.531,E2 13298.531} C_VEL
LIN {X 0,Y 330.394,Z 685.03,A -85,B 0,C 180,E1 13306.795,E2 13306.795} C_VEL
LIN {X 0,Y 330.908,Z 685.03,A -85,B 0,C 180,E1 13314.763,E2 13314.763} C_VEL
LIN {X 0,Y 331.28,Z 685.03,A -85,B 0,C 180,E1 13319.995,E2 13319.995} C_VEL
LIN {X 0,Y 330.701,Z 685.03,A -85,B 0,C 180,E1 13327.862,E2 13327.862} C_VEL
LIN {X 0,Y 330.232,Z 685.03,A -85,B 0,C 180,E1 13335.906,E2 13335.906} C_VEL
LIN {X 0,Y 329.777,Z 685.03,A -85,B 0,C 180,E1 13344.312,E2 13344.312} C_VEL
LIN {X 0,Y 329.537,Z 685.03,A -85,B 0,C 180,E1 13350.237,E2 13350.237} C_VEL
LIN {X 0,Y 329.394,Z 685.03,A -85,B 0,C 180,E1 13355.776,E2 13355.776} C_VEL
LIN {X 0,Y 331.524,Z 690.438,A -85,B 0,C 180,E1 13356.679,E2 13356.679} C_VEL
LIN {X 0,Y 334.15,Z 694.058,A -85,B 0,C 180,E1 13357.586,E2 13357.586} C_VEL
LIN {X 0,Y 346.385,Z 714.952,A -85,B 0,C 180,E1 13362.05,E2 13362.05} C_VEL
LIN {X 0,Y 357.181,Z 740.12,A -85,B 0,C 180,E1 13366.668,E2 13366.668} C_VEL
LIN {X 0,Y 364.689,Z 765.285,A -85,B 0,C 180,E1 13371.08,E2 13371.08} C_VEL
LIN {X 0,Y 366.698,Z 777.719,A -85,B 0,C 180,E1 13373.193,E2 13373.193} C_VEL
LIN {X 0,Y 358.23,Z 807.06,A -85,B 0,C 180,E1 13377.144,E2 13377.144} C_VEL
LIN {X 0,Y 350.203,Z 831.197,A -85,B 0,C 180,E1 13381.707,E2 13381.707} C_VEL
LIN {X 0,Y 343.097,Z 851.624,A -85,B 0,C 180,E1 13387.174,E2 13387.174} C_VEL
LIN {X 0,Y 337.957,Z 866.848,A -85,B 0,C 180,E1 13393.128,E2 13393.128} C_VEL
LIN {X 0,Y 334.92,Z 877.276,A -85,B 0,C 180,E1 13399.617,E2 13399.617} C_VEL
LIN {X 0,Y 333.78,Z 881.727,A -85,B 0,C 180,E1 13404.812,E2 13404.812} C_VEL
LIN {X 0,Y 333.449,Z 883.236,A -85,B 0,C 180,E1 13410,E2 13410} C_VEL
LIN {X 0,Y 333.822,Z 881.156,A -85,B 0,C 180,E1 13416.111,E2 13416.111} C_VEL
LIN {X 0,Y 335.835,Z 873.6,A -85,B 0,C 180,E1 13422.983,E2 13422.983} C_VEL
LIN {X 0,Y 339.948,Z 860.76,A -85,B 0,C 180,E1 13429.446,E2 13429.446} C_VEL
LIN {X 0,Y 346.386,Z 842.291,A -85,B 0,C 180,E1 13435.48,E2 13435.48} C_VEL
LIN {X 0,Y 354.37,Z 818.746,A -85,B 0,C 180,E1 13440.73,E2 13440.73} C_VEL
LIN {X 0,Y 362.575,Z 792.331,A -85,B 0,C 180,E1 13444.908,E2 13444.908} C_VEL
LIN {X 0,Y 366.892,Z 775.243,A -85,B 0,C 180,E1 13447.036,E2 13447.036} C_VEL
LIN {X 0,Y 360.447,Z 749.714,A -85,B 0,C 180,E1 13451.529,E2 13451.529} C_VEL
LIN {X 0,Y 350.437,Z 723.427,A -85,B 0,C 180,E1 13456.23,E2 13456.23} C_VEL
LIN {X 0,Y 336.875,Z 697.939,A -85,B 0,C 180,E1 13461.326,E2 13461.326} C_VEL
LIN {X 0,Y 331.693,Z 690.582,A -85,B 0,C 180,E1 13463.133,E2 13463.133} C_VEL
LIN {X 0,Y 329.419,Z 685.03,A -85,B 0,C 180,E1 13464.156,E2 13464.156} C_VEL
LIN {X 0,Y 329.622,Z 685.03,A -85,B 0,C 180,E1 13470.437,E2 13470.437} C_VEL
LIN {X 0,Y 329.938,Z 685.03,A -85,B 0,C 180,E1 13478.545,E2 13478.545} C_VEL
LIN {X 0,Y 330.509,Z 685.03,A -85,B 0,C 180,E1 13486.81,E2 13486.81} C_VEL
LIN {X 0,Y 330.911,Z 685.03,A -85,B 0,C 180,E1 13494.773,E2 13494.773} C_VEL
LIN {X 0,Y 331.265,Z 685.03,A -85,B 0,C 180,E1 13500.005,E2 13500.005} C_VEL
LIN {X 0,Y 330.91,Z 685.03,A -85,B 0,C 180,E1 13505.237,E2 13505.237} C_VEL
LIN {X 0,Y 330.362,Z 685.03,A -85,B 0,C 180,E1 13513.206,E2 13513.206} C_VEL
LIN {X 0,Y 329.894,Z 685.03,A -85,B 0,C 180,E1 13521.469,E2 13521.469} C_VEL
LIN {X 0,Y 329.512,Z 685.03,A -85,B 0,C 180,E1 13529.795,E2 13529.795} C_VEL
LIN {X 0,Y 331.492,Z 690.314,A -85,B 0,C 180,E1 13530.538,E2 13530.538} C_VEL
LIN {X 0,Y 334.512,Z 694.223,A -85,B 0,C 180,E1 13531.46,E2 13531.46} C_VEL
LIN {X 0,Y 351.816,Z 720.497,A -85,B 0,C 180,E1 13536.238,E2 13536.238} C_VEL
LIN {X 0,Y 368.273,Z 751.877,A -85,B 0,C 180,E1 13540.483,E2 13540.483} C_VEL
LIN {X 0,Y 377.503,Z 777.027,A -85,B 0,C 180,E1 13543.284,E2 13543.284} C_VEL
LIN {X 0,Y 370.045,Z 817.709,A -85,B 0,C 180,E1 13545.504,E2 13545.504} C_VEL
LIN {X 0,Y 361.616,Z 854.755,A -85,B 0,C 180,E1 13548.595,E2 13548.595} C_VEL
LIN {X 0,Y 352.85,Z 889.078,A -85,B 0,C 180,E1 13552.643,E2 13552.643} C_VEL
LIN {X 0,Y 344.897,Z 919.659,A -85,B 0,C 180,E1 13557.591,E2 13557.591} C_VEL
LIN {X 0,Y 338.819,Z 945.377,A -85,B 0,C 180,E1 13563.211,E2 13563.211} C_VEL
LIN {X 0,Y 334.677,Z 966.685,A -85,B 0,C 180,E1 13569.547,E2 13569.547} C_VEL
LIN {X 0,Y 332.779,Z 982.353,A -85,B 0,C 180,E1 13576.228,E2 13576.228} C_VEL
LIN {X 0,Y 332.452,Z 991.067,A -85,B 0,C 180,E1 13582.174,E2 13582.174} C_VEL
LIN {X 0,Y 332.522,Z 994.854,A -85,B 0,C 180,E1 13587.399,E2 13587.399} C_VEL
LIN {X 0,Y 332.55,Z 994.861,A -85,B 0,C 180,E1 13592.601,E2 13592.601} C_VEL
LIN {X 0,Y 332.432,Z 991.069,A -85,B 0,C 180,E1 13597.827,E2 13597.827} C_VEL
LIN {X 0,Y 332.818,Z 982.364,A -85,B 0,C 180,E1 13603.771,E2 13603.771} C_VEL
LIN {X 0,Y 334.361,Z 968.588,A -85,B 0,C 180,E1 13609.784,E2 13609.784} C_VEL
LIN {X 0,Y 338.447,Z 946.648,A -85,B 0,C 180,E1 13616.478,E2 13616.478} C_VEL
LIN {X 0,Y 341.016,Z 935.61,A -85,B 0,C 180,E1 13619.128,E2 13619.128} C_VEL
LIN {X 0,Y 339.809,Z 925.407,A -85,B 0,C 180,E1 13621.517,E2 13621.517} C_VEL
LIN {X 0,Y 338.935,Z 914.607,A -85,B 0,C 180,E1 13623.846,E2 13623.846} C_VEL
LIN {X 0,Y 347.928,Z 881.742,A -85,B 0,C 180,E1 13628.994,E2 13628.994} C_VEL
LIN {X 0,Y 357.232,Z 846.462,A -85,B 0,C 180,E1 13632.933,E2 13632.933} C_VEL
LIN {X 0,Y 365.534,Z 810.105,A -85,B 0,C 180,E1 13635.786,E2 13635.786} C_VEL
LIN {X 0,Y 371.416,Z 779.474,A -85,B 0,C 180,E1 13637.424,E2 13637.424} C_VEL
LIN {X 0,Y 361.576,Z 752.967,A -85,B 0,C 180,E1 13640.568,E2 13640.568} C_VEL
LIN {X 0,Y 345.509,Z 722.048,A -85,B 0,C 180,E1 13645.022,E2 13645.022} C_VEL
LIN {X 0,Y 329.2,Z 697.554,A -85,B 0,C 180,E1 13649.814,E2 13649.814} C_VEL
LIN {X 0,Y 324.701,Z 691.203,A -85,B 0,C 180,E1 13651.318,E2 13651.318} C_VEL
LIN {X 0,Y 321.816,Z 686.123,A -85,B 0,C 180,E1 13652.382,E2 13652.382} C_VEL
LIN {X 0,Y 321.742,Z 685.03,A -85,B 0,C 180,E1 13652.583,E2 13652.583} C_VEL
LIN {X 0,Y 322.078,Z 685.03,A -85,B 0,C 180,E1 13660.851,E2 13660.851} C_VEL
LIN {X 0,Y 322.59,Z 685.03,A -85,B 0,C 180,E1 13669.211,E2 13669.211} C_VEL
LIN {X 0,Y 323.205,Z 685.03,A -85,B 0,C 180,E1 13677.319,E2 13677.319} C_VEL
LIN {X 0,Y 323.271,Z 685.03,A -85,B 0,C 180,E1 13682.67,E2 13682.67} C_VEL
LIN {X 0,Y 322.611,Z 685.03,A -85,B 0,C 180,E1 13690.808,E2 13690.808} C_VEL
LIN {X 0,Y 322.088,Z 685.03,A -85,B 0,C 180,E1 13699.138,E2 13699.138} C_VEL
LIN {X 0,Y 321.72,Z 685.03,A -85,B 0,C 180,E1 13706.979,E2 13706.979} C_VEL
LIN {X 0,Y 321.482,Z 685.239,A -85,B 0,C 180,E1 13713.496,E2 13713.496} C_VEL
LIN {X 0,Y 323.656,Z 690.524,A -85,B 0,C 180,E1 13714.498,E2 13714.498} C_VEL
LIN {X 0,Y 326.165,Z 693.642,A -85,B 0,C 180,E1 13715.416,E2 13715.416} C_VEL
LIN {X 0,Y 338.562,Z 714.55,A -85,B 0,C 180,E1 13720.253,E2 13720.253} C_VEL
LIN {X 0,Y 348.768,Z 736.816,A -85,B 0,C 180,E1 13724.695,E2 13724.695} C_VEL
LIN {X 0,Y 357.111,Z 763.132,A -85,B 0,C 180,E1 13729.505,E2 13729.505} C_VEL
LIN {X 0,Y 360.191,Z 780.491,A -85,B 0,C 180,E1 13732.602,E2 13732.602} C_VEL
LIN {X 0,Y 351.511,Z 809.046,A -85,B 0,C 180,E1 13736.555,E2 13736.555} C_VEL
LIN {X 0,Y 342.877,Z 833.831,A -85,B 0,C 180,E1 13741.385,E2 13741.385} C_VEL
LIN {X 0,Y 335.911,Z 852.964,A -85,B 0,C 180,E1 13746.657,E2 13746.657} C_VEL
LIN {X 0,Y 330.487,Z 868.179,A -85,B 0,C 180,E1 13752.737,E2 13752.737} C_VEL
LIN {X 0,Y 327.248,Z 878.593,A -85,B 0,C 180,E1 13759.371,E2 13759.371} C_VEL
LIN {X 0,Y 326.017,Z 883.039,A -85,B 0,C 180,E1 13764.688,E2 13764.688} C_VEL
LIN {X 0,Y 325.67,Z 884.545,A -85,B 0,C 180,E1 13770,E2 13770} C_VEL
LIN {X 0,Y 325.981,Z 882.985,A -85,B 0,C 180,E1 13775.312,E2 13775.312} C_VEL
LIN {X 0,Y 327.727,Z 876.777,A -85,B 0,C 180,E1 13781.958,E2 13781.958} C_VEL
LIN {X 0,Y 331.514,Z 865.211,A -85,B 0,C 180,E1 13788.58,E2 13788.58} C_VEL
LIN {X 0,Y 337.672,Z 848.089,A -85,B 0,C 180,E1 13794.768,E2 13794.768} C_VEL
LIN {X 0,Y 345.521,Z 826.366,A -85,B 0,C 180,E1 13800.148,E2 13800.148} C_VEL
LIN {X 0,Y 354.334,Z 800.145,A -85,B 0,C 180,E1 13804.722,E2 13804.722} C_VEL
LIN {X 0,Y 360.364,Z 778.297,A -85,B 0,C 180,E1 13807.597,E2 13807.597} C_VEL
LIN {X 0,Y 353.913,Z 751.71,A -85,B 0,C 180,E1 13812.452,E2 13812.452} C_VEL
LIN {X 0,Y 344.08,Z 725.526,A -85,B 0,C 180,E1 13817.345,E2 13817.345} C_VEL
LIN {X 0,Y 331.942,Z 703.01,A -85,B 0,C 180,E1 13822.197,E2 13822.197} C_VEL
LIN {X 0,Y 324.263,Z 691.03,A -85,B 0,C 180,E1 13825.151,E2 13825.151} C_VEL
LIN {X 0,Y 321.582,Z 686.321,A -85,B 0,C 180,E1 13826.255,E2 13826.255} C_VEL
LIN {X 0,Y 321.505,Z 685.03,A -85,B 0,C 180,E1 13826.502,E2 13826.502} C_VEL
LIN {X 0,Y 321.757,Z 685.03,A -85,B 0,C 180,E1 13833.008,E2 13833.008} C_VEL
LIN {X 0,Y 322.142,Z 685.03,A -85,B 0,C 180,E1 13840.866,E2 13840.866} C_VEL
LIN {X 0,Y 322.57,Z 685.03,A -85,B 0,C 180,E1 13846.479,E2 13846.479} C_VEL
LIN {X 0,Y 322.982,Z 685.03,A -85,B 0,C 180,E1 13854.644,E2 13854.644} C_VEL
LIN {X 0,Y 323.361,Z 685.03,A -85,B 0,C 180,E1 13860.005,E2 13860.005} C_VEL
LIN {X 0,Y 322.98,Z 685.03,A -85,B 0,C 180,E1 13865.366,E2 13865.366} C_VEL
LIN {X 0,Y 322.417,Z 685.03,A -85,B 0,C 180,E1 13873.538,E2 13873.538} C_VEL
LIN {X 0,Y 321.96,Z 685.03,A -85,B 0,C 180,E1 13882.025,E2 13882.025} C_VEL
LIN {X 0,Y 321.663,Z 685.03,A -85,B 0,C 180,E1 13887.556,E2 13887.556} C_VEL
LIN {X 0,Y 323.712,Z 690.399,A -85,B 0,C 180,E1 13888.412,E2 13888.412} C_VEL
LIN {X 0,Y 326.622,Z 693.889,A -85,B 0,C 180,E1 13889.38,E2 13889.38} C_VEL
LIN {X 0,Y 342.707,Z 717.98,A -85,B 0,C 180,E1 13894.251,E2 13894.251} C_VEL
LIN {X 0,Y 358.967,Z 747.39,A -85,B 0,C 180,E1 13898.707,E2 13898.707} C_VEL
LIN {X 0,Y 370.998,Z 777.502,A -85,B 0,C 180,E1 13902.392,E2 13902.392} C_VEL
LIN {X 0,Y 363.953,Z 817.249,A -85,B 0,C 180,E1 13904.69,E2 13904.69} C_VEL
LIN {X 0,Y 355.012,Z 854.911,A -85,B 0,C 180,E1 13907.896,E2 13907.896} C_VEL
LIN {X 0,Y 346.064,Z 888.329,A -85,B 0,C 180,E1 13911.919,E2 13911.919} C_VEL
LIN {X 0,Y 337.929,Z 918.179,A -85,B 0,C 180,E1 13916.838,E2 13916.838} C_VEL
LIN {X 0,Y 331.376,Z 943.915,A -85,B 0,C 180,E1 13922.559,E2 13922.559} C_VEL
LIN {X 0,Y 326.981,Z 965.267,A -85,B 0,C 180,E1 13929.044,E2 13929.044} C_VEL
LIN {X 0,Y 325.093,Z 979.668,A -85,B 0,C 180,E1 13935.209,E2 13935.209} C_VEL
LIN {X 0,Y 324.669,Z 988.26,A -85,B 0,C 180,E1 13940.638,E2 13940.638} C_VEL
LIN {X 0,Y 324.687,Z 992.101,A -85,B 0,C 180,E1 13944.667,E2 13944.667} C_VEL
LIN {X 0,Y 324.864,Z 994.064,A -85,B 0,C 180,E1 13950,E2 13950} C_VEL
LIN {X 0,Y 324.696,Z 992.108,A -85,B 0,C 180,E1 13955.333,E2 13955.333} C_VEL
LIN {X 0,Y 324.784,Z 985.04,A -85,B 0,C 180,E1 13961.708,E2 13961.708} C_VEL
LIN {X 0,Y 325.968,Z 972.555,A -85,B 0,C 180,E1 13968.144,E2 13968.144} C_VEL
LIN {X 0,Y 329.464,Z 952.596,A -85,B 0,C 180,E1 13975.066,E2 13975.066} C_VEL
LIN {X 0,Y 335.491,Z 927.533,A -85,B 0,C 180,E1 13981.283,E2 13981.283} C_VEL
LIN {X 0,Y 338.935,Z 914.607,A -85,B 0,C 180,E1 13983.846,E2 13983.846} C_VEL
LIN {X 0,Y 338.567,Z 903.368,A -85,B 0,C 180,E1 13986.122,E2 13986.122} C_VEL
LIN {X 0,Y 338.218,Z 891.396,A -85,B 0,C 180,E1 13988.299,E2 13988.299} C_VEL
LIN {X 0,Y 347.923,Z 857.283,A -85,B 0,C 180,E1 13992.606,E2 13992.606} C_VEL
LIN {X 0,Y 357.263,Z 820.299,A -85,B 0,C 180,E1 13995.893,E2 13995.893} C_VEL
LIN {X 0,Y 364.96,Z 783.193,A -85,B 0,C 180,E1 13998.094,E2 13998.094} C_VEL
LIN {X 0,Y 362.504,Z 772.961,A -85,B 0,C 180,E1 13999.199,E2 13999.199} C_VEL
LIN {X 0,Y 348.805,Z 741.263,A -85,B 0,C 180,E1 14003.495,E2 14003.495} C_VEL
LIN {X 0,Y 334.093,Z 715.926,A -85,B 0,C 180,E1 14007.848,E2 14007.848} C_VEL
LIN {X 0,Y 321.411,Z 697.598,A -85,B 0,C 180,E1 14011.995,E2 14011.995} C_VEL
LIN {X 0,Y 317.363,Z 691.589,A -85,B 0,C 180,E1 14013.512,E2 14013.512} C_VEL
LIN {X 0,Y 314.08,Z 686.851,A -85,B 0,C 180,E1 14014.82,E2 14014.82} C_VEL
LIN {X 0,Y 313.883,Z 685.03,A -85,B 0,C 180,E1 14015.246,E2 14015.246} C_VEL
LIN {X 0,Y 314.377,Z 685.03,A -85,B 0,C 180,E1 14023.737,E2 14023.737} C_VEL
LIN {X 0,Y 314.837,Z 685.03,A -85,B 0,C 180,E1 14031.728,E2 14031.728} C_VEL
LIN {X 0,Y 315.476,Z 685.03,A -85,B 0,C 180,E1 14039.995,E2 14039.995} C_VEL
LIN {X 0,Y 315.057,Z 685.03,A -85,B 0,C 180,E1 14045.491,E2 14045.491} C_VEL
LIN {X 0,Y 314.481,Z 685.03,A -85,B 0,C 180,E1 14053.875,E2 14053.875} C_VEL
LIN {X 0,Y 314.139,Z 685.03,A -85,B 0,C 180,E1 14059.642,E2 14059.642} C_VEL
LIN {X 0,Y 313.807,Z 685.03,A -85,B 0,C 180,E1 14065.636,E2 14065.636} C_VEL
LIN {X 0,Y 313.625,Z 685.706,A -85,B 0,C 180,E1 14070.963,E2 14070.963} C_VEL
LIN {X 0,Y 316.205,Z 690.948,A -85,B 0,C 180,E1 14072.21,E2 14072.21} C_VEL
LIN {X 0,Y 318.497,Z 693.872,A -85,B 0,C 180,E1 14073.152,E2 14073.152} C_VEL
LIN {X 0,Y 330.215,Z 713.022,A -85,B 0,C 180,E1 14078.081,E2 14078.081} C_VEL
LIN {X 0,Y 341.621,Z 736.719,A -85,B 0,C 180,E1 14083.198,E2 14083.198} C_VEL
LIN {X 0,Y 350.261,Z 764.087,A -85,B 0,C 180,E1 14088.421,E2 14088.421} C_VEL
LIN {X 0,Y 353.833,Z 782.684,A -85,B 0,C 180,E1 14091.929,E2 14091.929} C_VEL
LIN {X 0,Y 344.621,Z 811.661,A -85,B 0,C 180,E1 14096.053,E2 14096.053} C_VEL
LIN {X 0,Y 335.889,Z 835.63,A -85,B 0,C 180,E1 14100.853,E2 14100.853} C_VEL
LIN {X 0,Y 328.122,Z 855.901,A -85,B 0,C 180,E1 14106.647,E2 14106.647} C_VEL
LIN {X 0,Y 322.533,Z 870.837,A -85,B 0,C 180,E1 14112.998,E2 14112.998} C_VEL
LIN {X 0,Y 319.586,Z 879.909,A -85,B 0,C 180,E1 14119.113,E2 14119.113} C_VEL
LIN {X 0,Y 318.27,Z 884.35,A -85,B 0,C 180,E1 14124.559,E2 14124.559} C_VEL
LIN {X 0,Y 317.887,Z 885.856,A -85,B 0,C 180,E1 14130,E2 14130} C_VEL
LIN {X 0,Y 318.216,Z 884.3,A -85,B 0,C 180,E1 14135.442,E2 14135.442} C_VEL
LIN {X 0,Y 320.066,Z 878.101,A -85,B 0,C 180,E1 14142.249,E2 14142.249} C_VEL
LIN {X 0,Y 324.115,Z 866.541,A -85,B 0,C 180,E1 14149.02,E2 14149.02} C_VEL
LIN {X 0,Y 330.581,Z 849.441,A -85,B 0,C 180,E1 14155.337,E2 14155.337} C_VEL
LIN {X 0,Y 338.806,Z 827.739,A -85,B 0,C 180,E1 14160.81,E2 14160.81} C_VEL
LIN {X 0,Y 347.974,Z 801.556,A -85,B 0,C 180,E1 14165.451,E2 14165.451} C_VEL
LIN {X 0,Y 353.903,Z 781.518,A -85,B 0,C 180,E1 14168.146,E2 14168.146} C_VEL
LIN {X 0,Y 347.691,Z 754.67,A -85,B 0,C 180,E1 14173.243,E2 14173.243} C_VEL
LIN {X 0,Y 338.671,Z 729.887,A -85,B 0,C 180,E1 14178.071,E2 14178.071} C_VEL
LIN {X 0,Y 327.842,Z 708.968,A -85,B 0,C 180,E1 14182.772,E2 14182.772} C_VEL
LIN {X 0,Y 320.366,Z 697.014,A -85,B 0,C 180,E1 14185.899,E2 14185.899} C_VEL
LIN {X 0,Y 316.72,Z 691.33,A -85,B 0,C 180,E1 14187.444,E2 14187.444} C_VEL
LIN {X 0,Y 313.757,Z 686.485,A -85,B 0,C 180,E1 14188.786,E2 14188.786} C_VEL
LIN {X 0,Y 313.633,Z 685.03,A -85,B 0,C 180,E1 14189.097,E2 14189.097} C_VEL
LIN {X 0,Y 313.985,Z 685.03,A -85,B 0,C 180,E1 14197.396,E2 14197.396} C_VEL
LIN {X 0,Y 314.462,Z 685.03,A -85,B 0,C 180,E1 14203.685,E2 14203.685} C_VEL
LIN {X 0,Y 314.874,Z 685.03,A -85,B 0,C 180,E1 14211.74,E2 14211.74} C_VEL
LIN {X 0,Y 315.463,Z 685.03,A -85,B 0,C 180,E1 14220.005,E2 14220.005} C_VEL
LIN {X 0,Y 315.06,Z 685.03,A -85,B 0,C 180,E1 14225.502,E2 14225.502} C_VEL
LIN {X 0,Y 314.451,Z 685.03,A -85,B 0,C 180,E1 14233.887,E2 14233.887} C_VEL
LIN {X 0,Y 314.104,Z 685.03,A -85,B 0,C 180,E1 14239.655,E2 14239.655} C_VEL
LIN {X 0,Y 313.862,Z 685.191,A -85,B 0,C 180,E1 14245.086,E2 14245.086} C_VEL
LIN {X 0,Y 315.808,Z 690.316,A -85,B 0,C 180,E1 14245.981,E2 14245.981} C_VEL
LIN {X 0,Y 318.85,Z 693.741,A -85,B 0,C 180,E1 14247.106,E2 14247.106} C_VEL
LIN {X 0,Y 334.922,Z 717.36,A -85,B 0,C 180,E1 14252.445,E2 14252.445} C_VEL
LIN {X 0,Y 351.048,Z 745.93,A -85,B 0,C 180,E1 14257.194,E2 14257.194} C_VEL
LIN {X 0,Y 363.759,Z 776.674,A -85,B 0,C 180,E1 14261.259,E2 14261.259} C_VEL
LIN {X 0,Y 364.867,Z 782.945,A -85,B 0,C 180,E1 14261.89,E2 14261.89} C_VEL
LIN {X 0,Y 356.848,Z 821.637,A -85,B 0,C 180,E1 14264.205,E2 14264.205} C_VEL
LIN {X 0,Y 347.337,Z 859.297,A -85,B 0,C 180,E1 14267.611,E2 14267.611} C_VEL
LIN {X 0,Y 337.57,Z 893.753,A -85,B 0,C 180,E1 14272.074,E2 14272.074} C_VEL
LIN {X 0,Y 328.963,Z 923.513,A -85,B 0,C 180,E1 14277.416,E2 14277.416} C_VEL
LIN {X 0,Y 322.695,Z 947.906,A -85,B 0,C 180,E1 14283.373,E2 14283.373} C_VEL
LIN {X 0,Y 318.697,Z 967.517,A -85,B 0,C 180,E1 14289.923,E2 14289.923} C_VEL
LIN {X 0,Y 317.073,Z 980.841,A -85,B 0,C 180,E1 14296.234,E2 14296.234} C_VEL
LIN {X 0,Y 316.823,Z 988.4,A -85,B 0,C 180,E1 14301.785,E2 14301.785} C_VEL
LIN {X 0,Y 316.95,Z 992.228,A -85,B 0,C 180,E1 14307.271,E2 14307.271} C_VEL
LIN {X 0,Y 316.961,Z 992.232,A -85,B 0,C 180,E1 14312.729,E2 14312.729} C_VEL
LIN {X 0,Y 316.8,Z 988.404,A -85,B 0,C 180,E1 14318.215,E2 14318.215} C_VEL
LIN {X 0,Y 317.175,Z 979.62,A -85,B 0,C 180,E1 14324.464,E2 14324.464} C_VEL
LIN {X 0,Y 318.973,Z 965.781,A -85,B 0,C 180,E1 14330.782,E2 14330.782} C_VEL
LIN {X 0,Y 323.447,Z 944.589,A -85,B 0,C 180,E1 14337.571,E2 14337.571} C_VEL
LIN {X 0,Y 330.367,Z 918.825,A -85,B 0,C 180,E1 14343.548,E2 14343.548} C_VEL
LIN {X 0,Y 338.218,Z 891.396,A -85,B 0,C 180,E1 14348.299,E2 14348.299} C_VEL
LIN {X 0,Y 338.363,Z 878.938,A -85,B 0,C 180,E1 14350.398,E2 14350.398} C_VEL
LIN {X 0,Y 338.933,Z 865.956,A -85,B 0,C 180,E1 14352.386,E2 14352.386} C_VEL
LIN {X 0,Y 348.771,Z 830.201,A -85,B 0,C 180,E1 14355.946,E2 14355.946} C_VEL
LIN {X 0,Y 357.335,Z 793.043,A -85,B 0,C 180,E1 14358.46,E2 14358.46} C_VEL
LIN {X 0,Y 358.886,Z 783.316,A -85,B 0,C 180,E1 14359.01,E2 14359.01} C_VEL
LIN {X 0,Y 347.101,Z 752.549,A -85,B 0,C 180,E1 14363.19,E2 14363.19} C_VEL
LIN {X 0,Y 332.862,Z 725.798,A -85,B 0,C 180,E1 14367.715,E2 14367.715} C_VEL
LIN {X 0,Y 318.92,Z 704.697,A -85,B 0,C 180,E1 14372.428,E2 14372.428} C_VEL
LIN {X 0,Y 313.006,Z 696.867,A -85,B 0,C 180,E1 14374.694,E2 14374.694} C_VEL
LIN {X 0,Y 309.941,Z 691.855,A -85,B 0,C 180,E1 14376.021,E2 14376.021} C_VEL
LIN {X 0,Y 306.392,Z 687.336,A -85,B 0,C 180,E1 14377.605,E2 14377.605} C_VEL
LIN {X 0,Y 306.037,Z 685.03,A -85,B 0,C 180,E1 14378.028,E2 14378.028} C_VEL
LIN {X 0,Y 306.546,Z 685.03,A -85,B 0,C 180,E1 14385.747,E2 14385.747} C_VEL
LIN {X 0,Y 307.123,Z 685.03,A -85,B 0,C 180,E1 14394.356,E2 14394.356} C_VEL
LIN {X 0,Y 307.573,Z 685.03,A -85,B 0,C 180,E1 14399.995,E2 14399.995} C_VEL
LIN {X 0,Y 307.124,Z 685.03,A -85,B 0,C 180,E1 14405.634,E2 14405.634} C_VEL
LIN {X 0,Y 306.745,Z 685.03,A -85,B 0,C 180,E1 14411.342,E2 14411.342} C_VEL
LIN {X 0,Y 306.321,Z 685.03,A -85,B 0,C 180,E1 14417.185,E2 14417.185} C_VEL
LIN {X 0,Y 306.005,Z 685.03,A -85,B 0,C 180,E1 14423.227,E2 14423.227} C_VEL
LIN {X 0,Y 305.72,Z 685.49,A -85,B 0,C 180,E1 14428.007,E2 14428.007} C_VEL
LIN {X 0,Y 307.972,Z 690.572,A -85,B 0,C 180,E1 14429.256,E2 14429.256} C_VEL
LIN {X 0,Y 310.739,Z 693.725,A -85,B 0,C 180,E1 14430.532,E2 14430.532} C_VEL
LIN {X 0,Y 322.691,Z 712.866,A -85,B 0,C 180,E1 14436.029,E2 14436.029} C_VEL
LIN {X 0,Y 333.959,Z 735.597,A -85,B 0,C 180,E1 14441.353,E2 14441.353} C_VEL
LIN {X 0,Y 342.367,Z 760.856,A -85,B 0,C 180,E1 14446.472,E2 14446.472} C_VEL
LIN {X 0,Y 347.415,Z 785.296,A -85,B 0,C 180,E1 14451.291,E2 14451.291} C_VEL
LIN {X 0,Y 338.33,Z 812.641,A -85,B 0,C 180,E1 14455.245,E2 14455.245} C_VEL
LIN {X 0,Y 329.12,Z 836.93,A -85,B 0,C 180,E1 14460.178,E2 14460.178} C_VEL
LIN {X 0,Y 320.908,Z 857.366,A -85,B 0,C 180,E1 14466.136,E2 14466.136} C_VEL
LIN {X 0,Y 315.048,Z 872.163,A -85,B 0,C 180,E1 14472.581,E2 14472.581} C_VEL
LIN {X 0,Y 311.92,Z 881.226,A -85,B 0,C 180,E1 14478.842,E2 14478.842} C_VEL
LIN {X 0,Y 310.517,Z 885.661,A -85,B 0,C 180,E1 14484.423,E2 14484.423} C_VEL
LIN {X 0,Y 310.11,Z 887.165,A -85,B 0,C 180,E1 14490,E2 14490} C_VEL
LIN {X 0,Y 310.466,Z 885.612,A -85,B 0,C 180,E1 14495.578,E2 14495.578} C_VEL
LIN {X 0,Y 312.414,Z 879.425,A -85,B 0,C 180,E1 14502.554,E2 14502.554} C_VEL
LIN {X 0,Y 316.735,Z 867.87,A -85,B 0,C 180,E1 14509.481,E2 14509.481} C_VEL
LIN {X 0,Y 323.557,Z 850.786,A -85,B 0,C 180,E1 14515.927,E2 14515.927} C_VEL
LIN {X 0,Y 332.137,Z 829.109,A -85,B 0,C 180,E1 14521.499,E2 14521.499} C_VEL
LIN {X 0,Y 341.69,Z 802.962,A -85,B 0,C 180,E1 14526.205,E2 14526.205} C_VEL
LIN {X 0,Y 347.354,Z 784.359,A -85,B 0,C 180,E1 14528.774,E2 14528.774} C_VEL
LIN {X 0,Y 341.724,Z 758.451,A -85,B 0,C 180,E1 14533.883,E2 14533.883} C_VEL
LIN {X 0,Y 333.75,Z 735.169,A -85,B 0,C 180,E1 14538.616,E2 14538.616} C_VEL
LIN {X 0,Y 323.021,Z 713.572,A -85,B 0,C 180,E1 14543.672,E2 14543.672} C_VEL
LIN {X 0,Y 313.247,Z 697.768,A -85,B 0,C 180,E1 14548.134,E2 14548.134} C_VEL
LIN {X 0,Y 309.246,Z 691.615,A -85,B 0,C 180,E1 14550.016,E2 14550.016} C_VEL
LIN {X 0,Y 305.872,Z 686.433,A -85,B 0,C 180,E1 14551.703,E2 14551.703} C_VEL
LIN {X 0,Y 305.755,Z 685.03,A -85,B 0,C 180,E1 14551.911,E2 14551.911} C_VEL
LIN {X 0,Y 306.185,Z 685.03,A -85,B 0,C 180,E1 14559.826,E2 14559.826} C_VEL
LIN {X 0,Y 306.651,Z 685.03,A -85,B 0,C 180,E1 14565.763,E2 14565.763} C_VEL
LIN {X 0,Y 306.932,Z 685.03,A -85,B 0,C 180,E1 14572.843,E2 14572.843} C_VEL
LIN {X 0,Y 307.559,Z 685.03,A -85,B 0,C 180,E1 14580.005,E2 14580.005} C_VEL
LIN {X 0,Y 307.126,Z 685.03,A -85,B 0,C 180,E1 14585.644,E2 14585.644} C_VEL
LIN {X 0,Y 306.679,Z 685.03,A -85,B 0,C 180,E1 14591.356,E2 14591.356} C_VEL
LIN {X 0,Y 306.296,Z 685.03,A -85,B 0,C 180,E1 14597.198,E2 14597.198} C_VEL
LIN {X 0,Y 306.057,Z 685.526,A -85,B 0,C 180,E1 14602.238,E2 14602.238} C_VEL
LIN {X 0,Y 308.36,Z 690.69,A -85,B 0,C 180,E1 14603.401,E2 14603.401} C_VEL
LIN {X 0,Y 311.104,Z 693.395,A -85,B 0,C 180,E1 14604.538,E2 14604.538} C_VEL
LIN {X 0,Y 325.41,Z 714.447,A -85,B 0,C 180,E1 14609.904,E2 14609.904} C_VEL
LIN {X 0,Y 340.378,Z 739.311,A -85,B 0,C 180,E1 14614.711,E2 14614.711} C_VEL
LIN {X 0,Y 353.713,Z 768.484,A -85,B 0,C 180,E1 14619.076,E2 14619.076} C_VEL
LIN {X 0,Y 358.889,Z 783.43,A -85,B 0,C 180,E1 14621.017,E2 14621.017} C_VEL
LIN {X 0,Y 350.514,Z 822.897,A -85,B 0,C 180,E1 14623.47,E2 14623.47} C_VEL
LIN {X 0,Y 340.439,Z 860.651,A -85,B 0,C 180,E1 14627.002,E2 14627.002} C_VEL
LIN {X 0,Y 330.402,Z 894.302,A -85,B 0,C 180,E1 14631.518,E2 14631.518} C_VEL
LIN {X 0,Y 321.393,Z 923.93,A -85,B 0,C 180,E1 14637.027,E2 14637.027} C_VEL
LIN {X 0,Y 314.962,Z 947.851,A -85,B 0,C 180,E1 14643.105,E2 14643.105} C_VEL
LIN {X 0,Y 310.698,Z 967.857,A -85,B 0,C 180,E1 14650.125,E2 14650.125} C_VEL
LIN {X 0,Y 309.165,Z 980.974,A -85,B 0,C 180,E1 14656.833,E2 14656.833} C_VEL
LIN {X 0,Y 308.97,Z 988.415,A -85,B 0,C 180,E1 14662.987,E2 14662.987} C_VEL
LIN {X 0,Y 309.153,Z 990.913,A -85,B 0,C 180,E1 14667.202,E2 14667.202} C_VEL
LIN {X 0,Y 309.164,Z 990.918,A -85,B 0,C 180,E1 14672.798,E2 14672.798} C_VEL
LIN {X 0,Y 308.97,Z 987.068,A -85,B 0,C 180,E1 14678.425,E2 14678.425} C_VEL
LIN {X 0,Y 309.364,Z 978.249,A -85,B 0,C 180,E1 14684.838,E2 14684.838} C_VEL
LIN {X 0,Y 311.295,Z 964.377,A -85,B 0,C 180,E1 14691.319,E2 14691.319} C_VEL
LIN {X 0,Y 315.951,Z 943.671,A -85,B 0,C 180,E1 14698.128,E2 14698.128} C_VEL
LIN {X 0,Y 323.434,Z 917.456,A -85,B 0,C 180,E1 14704.342,E2 14704.342} C_VEL
LIN {X 0,Y 332.666,Z 886.816,A -85,B 0,C 180,E1 14709.634,E2 14709.634} C_VEL
LIN {X 0,Y 338.933,Z 865.956,A -85,B 0,C 180,E1 14712.386,E2 14712.386} C_VEL
LIN {X 0,Y 339.566,Z 852.491,A -85,B 0,C 180,E1 14714.284,E2 14714.284} C_VEL
LIN {X 0,Y 339.987,Z 840.408,A -85,B 0,C 180,E1 14715.878,E2 14715.878} C_VEL
LIN {X 0,Y 340.463,Z 838.535,A -85,B 0,C 180,E1 14716.059,E2 14716.059} C_VEL
LIN {X 0,Y 350.212,Z 799.604,A -85,B 0,C 180,E1 14718.986,E2 14718.986} C_VEL
LIN {X 0,Y 352.615,Z 785.55,A -85,B 0,C 180,E1 14719.84,E2 14719.84} C_VEL
LIN {X 0,Y 341.105,Z 755.129,A -85,B 0,C 180,E1 14724.21,E2 14724.21} C_VEL
LIN {X 0,Y 327.795,Z 729.35,A -85,B 0,C 180,E1 14728.806,E2 14728.806} C_VEL
LIN {X 0,Y 312.285,Z 705.71,A -85,B 0,C 180,E1 14734.506,E2 14734.506} C_VEL
LIN {X 0,Y 306.278,Z 697.922,A -85,B 0,C 180,E1 14737.071,E2 14737.071} C_VEL
LIN {X 0,Y 302.317,Z 691.992,A -85,B 0,C 180,E1 14739.005,E2 14739.005} C_VEL
LIN {X 0,Y 298.524,Z 687.218,A -85,B 0,C 180,E1 14741.005,E2 14741.005} C_VEL
LIN {X 0,Y 298.249,Z 685.03,A -85,B 0,C 180,E1 14741.561,E2 14741.561} C_VEL
LIN {X 0,Y 298.731,Z 685.03,A -85,B 0,C 180,E1 14748.338,E2 14748.338} C_VEL
LIN {X 0,Y 299.483,Z 685.03,A -85,B 0,C 180,E1 14757.107,E2 14757.107} C_VEL
LIN {X 0,Y 299.546,Z 685.03,A -85,B 0,C 180,E1 14762.882,E2 14762.882} C_VEL
LIN {X 0,Y 298.783,Z 685.03,A -85,B 0,C 180,E1 14771.649,E2 14771.649} C_VEL
LIN {X 0,Y 298.362,Z 685.03,A -85,B 0,C 180,E1 14777.658,E2 14777.658} C_VEL
LIN {X 0,Y 297.91,Z 685.03,A -85,B 0,C 180,E1 14784.506,E2 14784.506} C_VEL
LIN {X 0,Y 299.553,Z 689.9,A -85,B 0,C 180,E1 14785.65,E2 14785.65} C_VEL
LIN {X 0,Y 303.039,Z 693.523,A -85,B 0,C 180,E1 14787.518,E2 14787.518} C_VEL
LIN {X 0,Y 308.574,Z 702.393,A -85,B 0,C 180,E1 14790.479,E2 14790.479} C_VEL
LIN {X 0,Y 316.323,Z 714.959,A -85,B 0,C 180,E1 14794.34,E2 14794.34} C_VEL
LIN {X 0,Y 326.676,Z 735.506,A -85,B 0,C 180,E1 14799.576,E2 14799.576} C_VEL
LIN {X 0,Y 334.652,Z 757.805,A -85,B 0,C 180,E1 14804.418,E2 14804.418} C_VEL
LIN {X 0,Y 340.161,Z 782.701,A -85,B 0,C 180,E1 14809.523,E2 14809.523} C_VEL
LIN {X 0,Y 340.208,Z 790.461,A -85,B 0,C 180,E1 14810.948,E2 14810.948} C_VEL
LIN {X 0,Y 330.204,Z 818.83,A -85,B 0,C 180,E1 14815.329,E2 14815.329} C_VEL
LIN {X 0,Y 320.376,Z 843.066,A -85,B 0,C 180,E1 14820.709,E2 14820.709} C_VEL
LIN {X 0,Y 312.241,Z 862.153,A -85,B 0,C 180,E1 14826.874,E2 14826.874} C_VEL
LIN {X 0,Y 306.326,Z 876.519,A -85,B 0,C 180,E1 14833.937,E2 14833.937} C_VEL
LIN {X 0,Y 303.269,Z 885.151,A -85,B 0,C 180,E1 14841.415,E2 14841.415} C_VEL
LIN {X 0,Y 302.531,Z 888.069,A -85,B 0,C 180,E1 14847.141,E2 14847.141} C_VEL
LIN {X 0,Y 302.556,Z 887.639,A -85,B 0,C 180,E1 14854.189,E2 14854.189} C_VEL
LIN {X 0,Y 304.28,Z 882.426,A -85,B 0,C 180,E1 14861.442,E2 14861.442} C_VEL
LIN {X 0,Y 308.16,Z 871.962,A -85,B 0,C 180,E1 14868.56,E2 14868.56} C_VEL
LIN {X 0,Y 314.434,Z 856.95,A -85,B 0,C 180,E1 14874.948,E2 14874.948} C_VEL
LIN {X 0,Y 323.169,Z 836.24,A -85,B 0,C 180,E1 14880.906,E2 14880.906} C_VEL
LIN {X 0,Y 333.333,Z 810.316,A -85,B 0,C 180,E1 14886.051,E2 14886.051} C_VEL
LIN {X 0,Y 340.875,Z 787.74,A -85,B 0,C 180,E1 14889.317,E2 14889.317} C_VEL
LIN {X 0,Y 336.012,Z 762.995,A -85,B 0,C 180,E1 14894.387,E2 14894.387} C_VEL
LIN {X 0,Y 328.347,Z 739.311,A -85,B 0,C 180,E1 14899.412,E2 14899.412} C_VEL
LIN {X 0,Y 317.565,Z 716.954,A -85,B 0,C 180,E1 14904.933,E2 14904.933} C_VEL
LIN {X 0,Y 306.636,Z 698.804,A -85,B 0,C 180,E1 14910.428,E2 14910.428} C_VEL
LIN {X 0,Y 302.866,Z 692.735,A -85,B 0,C 180,E1 14912.448,E2 14912.448} C_VEL
LIN {X 0,Y 298.247,Z 687.324,A -85,B 0,C 180,E1 14914.96,E2 14914.96} C_VEL
LIN {X 0,Y 297.964,Z 685.03,A -85,B 0,C 180,E1 14915.485,E2 14915.485} C_VEL
LIN {X 0,Y 298.512,Z 685.03,A -85,B 0,C 180,E1 14923.834,E2 14923.834} C_VEL
LIN {X 0,Y 299.01,Z 685.03,A -85,B 0,C 180,E1 14931.298,E2 14931.298} C_VEL
LIN {X 0,Y 299.665,Z 685.03,A -85,B 0,C 180,E1 14940.006,E2 14940.006} C_VEL
LIN {X 0,Y 299.19,Z 685.03,A -85,B 0,C 180,E1 14945.794,E2 14945.794} C_VEL
LIN {X 0,Y 298.539,Z 685.03,A -85,B 0,C 180,E1 14954.644,E2 14954.644} C_VEL
LIN {X 0,Y 298.221,Z 685.372,A -85,B 0,C 180,E1 14958.823,E2 14958.823} C_VEL
LIN {X 0,Y 300.165,Z 690.242,A -85,B 0,C 180,E1 14960.032,E2 14960.032} C_VEL
LIN {X 0,Y 303.749,Z 693.938,A -85,B 0,C 180,E1 14961.784,E2 14961.784} C_VEL
LIN {X 0,Y 313.88,Z 708.466,A -85,B 0,C 180,E1 14966.216,E2 14966.216} C_VEL
LIN {X 0,Y 327.668,Z 729.432,A -85,B 0,C 180,E1 14971.208,E2 14971.208} C_VEL
LIN {X 0,Y 342.198,Z 757.596,A -85,B 0,C 180,E1 14976.194,E2 14976.194} C_VEL
LIN {X 0,Y 352.759,Z 786.071,A -85,B 0,C 180,E1 14980.244,E2 14980.244} C_VEL
LIN {X 0,Y 343.871,Z 825.45,A -85,B 0,C 180,E1 14982.817,E2 14982.817} C_VEL
LIN {X 0,Y 333.541,Z 861.997,A -85,B 0,C 180,E1 14986.377,E2 14986.377} C_VEL
LIN {X 0,Y 323.742,Z 893.391,A -85,B 0,C 180,E1 14990.699,E2 14990.699} C_VEL
LIN {X 0,Y 314.613,Z 922.05,A -85,B 0,C 180,E1 14996.112,E2 14996.112} C_VEL
LIN {X 0,Y 307.654,Z 946.168,A -85,B 0,C 180,E1 15002.331,E2 15002.331} C_VEL
LIN {X 0,Y 303.326,Z 964.711,A -85,B 0,C 180,E1 15008.858,E2 15008.858} C_VEL
LIN {X 0,Y 301.451,Z 978.111,A -85,B 0,C 180,E1 15015.505,E2 15015.505} C_VEL
LIN {X 0,Y 301.19,Z 985.731,A -85,B 0,C 180,E1 15021.356,E2 15021.356} C_VEL
LIN {X 0,Y 301.352,Z 989.597,A -85,B 0,C 180,E1 15027.13,E2 15027.13} C_VEL
LIN {X 0,Y 301.36,Z 989.602,A -85,B 0,C 180,E1 15032.87,E2 15032.87} C_VEL
LIN {X 0,Y 301.166,Z 985.737,A -85,B 0,C 180,E1 15038.645,E2 15038.645} C_VEL
LIN {X 0,Y 301.583,Z 976.882,A -85,B 0,C 180,E1 15045.23,E2 15045.23} C_VEL
LIN {X 0,Y 304.064,Z 961.053,A -85,B 0,C 180,E1 15052.62,E2 15052.62} C_VEL
LIN {X 0,Y 309.442,Z 939.545,A -85,B 0,C 180,E1 15059.587,E2 15059.587} C_VEL
LIN {X 0,Y 317.264,Z 913.82,A -85,B 0,C 180,E1 15065.628,E2 15065.628} C_VEL
LIN {X 0,Y 327.059,Z 883.076,A -85,B 0,C 180,E1 15070.888,E2 15070.888} C_VEL
LIN {X 0,Y 337.512,Z 848.922,A -85,B 0,C 180,E1 15075.059,E2 15075.059} C_VEL
LIN {X 0,Y 340.463,Z 838.535,A -85,B 0,C 180,E1 15076.059,E2 15076.059} C_VEL
LIN {X 0,Y 341.464,Z 824.165,A -85,B 0,C 180,E1 15077.744,E2 15077.744} C_VEL
LIN {X 0,Y 341.786,Z 811.24,A -85,B 0,C 180,E1 15079.139,E2 15079.139} C_VEL
LIN {X 0,Y 342.181,Z 809.259,A -85,B 0,C 180,E1 15079.28,E2 15079.28} C_VEL
LIN {X 0,Y 346.675,Z 788.745,A -85,B 0,C 180,E1 15080.546,E2 15080.546} C_VEL
LIN {X 0,Y 335.46,Z 758.003,A -85,B 0,C 180,E1 15085.186,E2 15085.186} C_VEL
LIN {X 0,Y 323.039,Z 733.903,A -85,B 0,C 180,E1 15089.757,E2 15089.757} C_VEL
LIN {X 0,Y 309.487,Z 712.425,A -85,B 0,C 180,E1 15095.128,E2 15095.128} C_VEL
LIN {X 0,Y 299.845,Z 699.048,A -85,B 0,C 180,E1 15099.657,E2 15099.657} C_VEL
LIN {X 0,Y 296.037,Z 693.509,A -85,B 0,C 180,E1 15101.803,E2 15101.803} C_VEL
LIN {X 0,Y 291.052,Z 687.536,A -85,B 0,C 180,E1 15104.971,E2 15104.971} C_VEL
LIN {X 0,Y 290.663,Z 685.03,A -85,B 0,C 180,E1 15105.527,E2 15105.527} C_VEL
LIN {X 0,Y 291.251,Z 685.03,A -85,B 0,C 180,E1 15114.047,E2 15114.047} C_VEL
LIN {X 0,Y 291.772,Z 685.03,A -85,B 0,C 180,E1 15119.994,E2 15119.994} C_VEL
LIN {X 0,Y 291.254,Z 685.03,A -85,B 0,C 180,E1 15125.942,E2 15125.942} C_VEL
LIN {X 0,Y 290.828,Z 685.03,A -85,B 0,C 180,E1 15131.972,E2 15131.972} C_VEL
LIN {X 0,Y 290.26,Z 685.14,A -85,B 0,C 180,E1 15140.274,E2 15140.274} C_VEL
LIN {X 0,Y 292.14,Z 690.326,A -85,B 0,C 180,E1 15141.885,E2 15141.885} C_VEL
LIN {X 0,Y 295.528,Z 693.302,A -85,B 0,C 180,E1 15144.002,E2 15144.002} C_VEL
LIN {X 0,Y 298.941,Z 698.848,A -85,B 0,C 180,E1 15146.203,E2 15146.203} C_VEL
LIN {X 0,Y 308.323,Z 713.448,A -85,B 0,C 180,E1 15151.509,E2 15151.509} C_VEL
LIN {X 0,Y 319.47,Z 735.055,A -85,B 0,C 180,E1 15157.604,E2 15157.604} C_VEL
LIN {X 0,Y 327.673,Z 757.545,A -85,B 0,C 180,E1 15162.816,E2 15162.816} C_VEL
LIN {X 0,Y 333.293,Z 782.335,A -85,B 0,C 180,E1 15168.138,E2 15168.138} C_VEL
LIN {X 0,Y 334.168,Z 792.063,A -85,B 0,C 180,E1 15170.132,E2 15170.132} C_VEL
LIN {X 0,Y 323.834,Z 820.21,A -85,B 0,C 180,E1 15174.546,E2 15174.546} C_VEL
LIN {X 0,Y 313.606,Z 844.352,A -85,B 0,C 180,E1 15179.992,E2 15179.992} C_VEL
LIN {X 0,Y 305.12,Z 863.36,A -85,B 0,C 180,E1 15186.247,E2 15186.247} C_VEL
LIN {X 0,Y 299.003,Z 877.459,A -85,B 0,C 180,E1 15193.295,E2 15193.295} C_VEL
LIN {X 0,Y 295.986,Z 885.242,A -85,B 0,C 180,E1 15199.721,E2 15199.721} C_VEL
LIN {X 0,Y 294.763,Z 889.378,A -85,B 0,C 180,E1 15207.066,E2 15207.066} C_VEL
LIN {X 0,Y 294.774,Z 889.342,A -85,B 0,C 180,E1 15212.934,E2 15212.934} C_VEL
LIN {X 0,Y 296.028,Z 885.133,A -85,B 0,C 180,E1 15220.277,E2 15220.277} C_VEL
LIN {X 0,Y 299.643,Z 875.829,A -85,B 0,C 180,E1 15227.587,E2 15227.587} C_VEL
LIN {X 0,Y 306.305,Z 860.709,A -85,B 0,C 180,E1 15234.7,E2 15234.7} C_VEL
LIN {X 0,Y 314.859,Z 841.462,A -85,B 0,C 180,E1 15240.669,E2 15240.669} C_VEL
LIN {X 0,Y 324.842,Z 817.349,A -85,B 0,C 180,E1 15245.867,E2 15245.867} C_VEL
LIN {X 0,Y 334.345,Z 791.073,A -85,B 0,C 180,E1 15249.905,E2 15249.905} C_VEL
LIN {X 0,Y 330.047,Z 766.384,A -85,B 0,C 180,E1 15255.145,E2 15255.145} C_VEL
LIN {X 0,Y 322.582,Z 742.713,A -85,B 0,C 180,E1 15260.415,E2 15260.415} C_VEL
LIN {X 0,Y 313.04,Z 722.189,A -85,B 0,C 180,E1 15265.76,E2 15265.76} C_VEL
LIN {X 0,Y 303.444,Z 705.582,A -85,B 0,C 180,E1 15271.006,E2 15271.006} C_VEL
LIN {X 0,Y 298.495,Z 698.431,A -85,B 0,C 180,E1 15273.856,E2 15273.856} C_VEL
LIN {X 0,Y 295.436,Z 692.875,A -85,B 0,C 180,E1 15275.89,E2 15275.89} C_VEL
LIN {X 0,Y 290.781,Z 687.843,A -85,B 0,C 180,E1 15278.92,E2 15278.92} C_VEL
LIN {X 0,Y 290.306,Z 685.03,A -85,B 0,C 180,E1 15279.481,E2 15279.481} C_VEL
LIN {X 0,Y 290.894,Z 685.03,A -85,B 0,C 180,E1 15288.031,E2 15288.031} C_VEL
LIN {X 0,Y 291.516,Z 685.03,A -85,B 0,C 180,E1 15297.039,E2 15297.039} C_VEL
LIN {X 0,Y 291.621,Z 685.03,A -85,B 0,C 180,E1 15302.972,E2 15302.972} C_VEL
LIN {X 0,Y 290.779,Z 685.03,A -85,B 0,C 180,E1 15311.985,E2 15311.985} C_VEL
LIN {X 0,Y 290.663,Z 685.573,A -85,B 0,C 180,E1 15314.761,E2 15314.761} C_VEL
LIN {X 0,Y 292.565,Z 690.321,A -85,B 0,C 180,E1 15316.247,E2 15316.247} C_VEL
LIN {X 0,Y 296.02,Z 693.544,A -85,B 0,C 180,E1 15318.294,E2 15318.294} C_VEL
LIN {X 0,Y 300.207,Z 699.329,A -85,B 0,C 180,E1 15320.605,E2 15320.605} C_VEL
LIN {X 0,Y 311.384,Z 715.621,A -85,B 0,C 180,E1 15325.766,E2 15325.766} C_VEL
LIN {X 0,Y 324.576,Z 736.844,A -85,B 0,C 180,E1 15330.87,E2 15330.87} C_VEL
LIN {X 0,Y 337.675,Z 763.593,A -85,B 0,C 180,E1 15335.736,E2 15335.736} C_VEL
LIN {X 0,Y 346.627,Z 788.697,A -85,B 0,C 180,E1 15339.463,E2 15339.463} C_VEL
LIN {X 0,Y 337.462,Z 827.034,A -85,B 0,C 180,E1 15342.069,E2 15342.069} C_VEL
LIN {X 0,Y 326.766,Z 863.096,A -85,B 0,C 180,E1 15345.697,E2 15345.697} C_VEL
LIN {X 0,Y 316.097,Z 895.564,A -85,B 0,C 180,E1 15350.355,E2 15350.355} C_VEL
LIN {X 0,Y 306.17,Z 925.348,A -85,B 0,C 180,E1 15356.326,E2 15356.326} C_VEL
LIN {X 0,Y 298.745,Z 950.272,A -85,B 0,C 180,E1 15363.366,E2 15363.366} C_VEL
LIN {X 0,Y 294.927,Z 967.258,A -85,B 0,C 180,E1 15370.019,E2 15370.019} C_VEL
LIN {X 0,Y 293.424,Z 980.546,A -85,B 0,C 180,E1 15377.725,E2 15377.725} C_VEL
LIN {X 0,Y 293.386,Z 986.798,A -85,B 0,C 180,E1 15384.096,E2 15384.096} C_VEL
LIN {X 0,Y 293.726,Z 988.822,A -85,B 0,C 180,E1 15390,E2 15390} C_VEL
LIN {X 0,Y 293.389,Z 986.806,A -85,B 0,C 180,E1 15395.904,E2 15395.904} C_VEL
LIN {X 0,Y 293.467,Z 980.513,A -85,B 0,C 180,E1 15402.314,E2 15402.314} C_VEL
LIN {X 0,Y 294.916,Z 967.228,A -85,B 0,C 180,E1 15410.004,E2 15410.004} C_VEL
LIN {X 0,Y 299.405,Z 947.913,A -85,B 0,C 180,E1 15417.431,E2 15417.431} C_VEL
LIN {X 0,Y 306.648,Z 923.805,A -85,B 0,C 180,E1 15424.039,E2 15424.039} C_VEL
LIN {X 0,Y 316.524,Z 894.224,A -85,B 0,C 180,E1 15429.885,E2 15429.885} C_VEL
LIN {X 0,Y 327.214,Z 861.928,A -85,B 0,C 180,E1 15434.45,E2 15434.45} C_VEL
LIN {X 0,Y 337.762,Z 826.255,A -85,B 0,C 180,E1 15438.002,E2 15438.002} C_VEL
LIN {X 0,Y 342.181,Z 809.259,A -85,B 0,C 180,E1 15439.28,E2 15439.28} C_VEL
LIN {X 0,Y 342.616,Z 797.877,A -85,B 0,C 180,E1 15440.386,E2 15440.386} C_VEL
LIN {X 0,Y 337.451,Z 781.346,A -85,B 0,C 180,E1 15442.862,E2 15442.862} C_VEL
LIN {X 0,Y 326.195,Z 753.166,A -85,B 0,C 180,E1 15447.627,E2 15447.627} C_VEL
LIN {X 0,Y 313.402,Z 729.886,A -85,B 0,C 180,E1 15452.776,E2 15452.776} C_VEL
LIN {X 0,Y 301.886,Z 712.339,A -85,B 0,C 180,E1 15457.978,E2 15457.978} C_VEL
LIN {X 0,Y 296.723,Z 705.319,A -85,B 0,C 180,E1 15460.693,E2 15460.693} C_VEL
LIN {X 0,Y 292.685,Z 699.352,A -85,B 0,C 180,E1 15463.137,E2 15463.137} C_VEL
LIN {X 0,Y 288.87,Z 693.772,A -85,B 0,C 180,E1 15465.821,E2 15465.821} C_VEL
LIN {X 0,Y 283.481,Z 687.643,A -85,B 0,C 180,E1 15470.5,E2 15470.5} C_VEL
LIN {X 0,Y 283.123,Z 685.03,A -85,B 0,C 180,E1 15471.18,E2 15471.18} C_VEL
LIN {X 0,Y 283.867,Z 685.03,A -85,B 0,C 180,E1 15479.994,E2 15479.994} C_VEL
LIN {X 0,Y 283.324,Z 685.03,A -85,B 0,C 180,E1 15486.108,E2 15486.108} C_VEL
LIN {X 0,Y 282.712,Z 685.48,A -85,B 0,C 180,E1 15494.383,E2 15494.383} C_VEL
LIN {X 0,Y 284.771,Z 690.611,A -85,B 0,C 180,E1 15496.923,E2 15496.923} C_VEL
LIN {X 0,Y 288.35,Z 693.532,A -85,B 0,C 180,E1 15499.852,E2 15499.852} C_VEL
LIN {X 0,Y 291.486,Z 699.02,A -85,B 0,C 180,E1 15502.437,E2 15502.437} C_VEL
LIN {X 0,Y 293.419,Z 701.625,A -85,B 0,C 180,E1 15503.782,E2 15503.782} C_VEL
LIN {X 0,Y 298.587,Z 709.896,A -85,B 0,C 180,E1 15507.25,E2 15507.25} C_VEL
LIN {X 0,Y 305.703,Z 721.914,A -85,B 0,C 180,E1 15511.544,E2 15511.544} C_VEL
LIN {X 0,Y 315.141,Z 741.268,A -85,B 0,C 180,E1 15517.185,E2 15517.185} C_VEL
LIN {X 0,Y 322.589,Z 763.792,A -85,B 0,C 180,E1 15522.605,E2 15522.605} C_VEL
LIN {X 0,Y 327.362,Z 788.074,A -85,B 0,C 180,E1 15528,E2 15528} C_VEL
LIN {X 0,Y 327.595,Z 795.381,A -85,B 0,C 180,E1 15529.505,E2 15529.505} C_VEL
LIN {X 0,Y 316.565,Z 823.805,A -85,B 0,C 180,E1 15534.173,E2 15534.173} C_VEL
LIN {X 0,Y 306.874,Z 845.695,A -85,B 0,C 180,E1 15539.264,E2 15539.264} C_VEL
LIN {X 0,Y 297.885,Z 864.917,A -85,B 0,C 180,E1 15545.736,E2 15545.736} C_VEL
LIN {X 0,Y 291.277,Z 879.355,A -85,B 0,C 180,E1 15553.216,E2 15553.216} C_VEL
LIN {X 0,Y 287.833,Z 887.781,A -85,B 0,C 180,E1 15560.951,E2 15560.951} C_VEL
LIN {X 0,Y 286.867,Z 890.885,A -85,B 0,C 180,E1 15567.814,E2 15567.814} C_VEL
LIN {X 0,Y 287.001,Z 890.653,A -85,B 0,C 180,E1 15573.014,E2 15573.014} C_VEL
LIN {X 0,Y 288.35,Z 886.45,A -85,B 0,C 180,E1 15580.554,E2 15580.554} C_VEL
LIN {X 0,Y 292.198,Z 877.153,A -85,B 0,C 180,E1 15588.051,E2 15588.051} C_VEL
LIN {X 0,Y 299.283,Z 861.917,A -85,B 0,C 180,E1 15595.375,E2 15595.375} C_VEL
LIN {X 0,Y 308.543,Z 841.972,A -85,B 0,C 180,E1 15601.624,E2 15601.624} C_VEL
LIN {X 0,Y 319.077,Z 817.463,A -85,B 0,C 180,E1 15606.917,E2 15606.917} C_VEL
LIN {X 0,Y 327.901,Z 792.648,A -85,B 0,C 180,E1 15610.853,E2 15610.853} C_VEL
LIN {X 0,Y 323.642,Z 767.822,A -85,B 0,C 180,E1 15616.358,E2 15616.358} C_VEL
LIN {X 0,Y 316.537,Z 745.064,A -85,B 0,C 180,E1 15621.713,E2 15621.713} C_VEL
LIN {X 0,Y 307.376,Z 724.767,A -85,B 0,C 180,E1 15627.324,E2 15627.324} C_VEL
LIN {X 0,Y 296.793,Z 706.358,A -85,B 0,C 180,E1 15633.796,E2 15633.796} C_VEL
LIN {X 0,Y 292.988,Z 700.323,A -85,B 0,C 180,E1 15636.382,E2 15636.382} C_VEL
LIN {X 0,Y 288.594,Z 694.459,A -85,B 0,C 180,E1 15639.652,E2 15639.652} C_VEL
LIN {X 0,Y 287.654,Z 692.472,A -85,B 0,C 180,E1 15640.477,E2 15640.477} C_VEL
LIN {X 0,Y 283.234,Z 687.89,A -85,B 0,C 180,E1 15644.461,E2 15644.461} C_VEL
LIN {X 0,Y 282.797,Z 685.03,A -85,B 0,C 180,E1 15645.325,E2 15645.325} C_VEL
LIN {X 0,Y 283.336,Z 685.03,A -85,B 0,C 180,E1 15653.892,E2 15653.892} C_VEL
LIN {X 0,Y 283.855,Z 685.03,A -85,B 0,C 180,E1 15660.006,E2 15660.006} C_VEL
LIN {X 0,Y 283.124,Z 685.03,A -85,B 0,C 180,E1 15667.662,E2 15667.662} C_VEL
LIN {X 0,Y 283.109,Z 685.406,A -85,B 0,C 180,E1 15669.11,E2 15669.11} C_VEL
LIN {X 0,Y 284.798,Z 690.191,A -85,B 0,C 180,E1 15671.099,E2 15671.099} C_VEL
LIN {X 0,Y 288.709,Z 693.42,A -85,B 0,C 180,E1 15674.187,E2 15674.187} C_VEL
LIN {X 0,Y 292.214,Z 699.037,A -85,B 0,C 180,E1 15676.698,E2 15676.698} C_VEL
LIN {X 0,Y 294.348,Z 701.787,A -85,B 0,C 180,E1 15678.015,E2 15678.015} C_VEL
LIN {X 0,Y 300.234,Z 710.193,A -85,B 0,C 180,E1 15681.278,E2 15681.278} C_VEL
LIN {X 0,Y 309.77,Z 724.164,A -85,B 0,C 180,E1 15685.716,E2 15685.716} C_VEL
LIN {X 0,Y 323.033,Z 747.115,A -85,B 0,C 180,E1 15691.187,E2 15691.187} C_VEL
LIN {X 0,Y 335.061,Z 774.596,A -85,B 0,C 180,E1 15696.108,E2 15696.108} C_VEL
LIN {X 0,Y 340.416,Z 793.043,A -85,B 0,C 180,E1 15698.803,E2 15698.803} C_VEL
LIN {X 0,Y 330.513,Z 830.784,A -85,B 0,C 180,E1 15701.478,E2 15701.478} C_VEL
LIN {X 0,Y 318.794,Z 867.868,A -85,B 0,C 180,E1 15705.447,E2 15705.447} C_VEL
LIN {X 0,Y 307.643,Z 899.816,A -85,B 0,C 180,E1 15710.383,E2 15710.383} C_VEL
LIN {X 0,Y 298.229,Z 926.827,A -85,B 0,C 180,E1 15716.18,E2 15716.18} C_VEL
LIN {X 0,Y 291.023,Z 949.939,A -85,B 0,C 180,E1 15723.019,E2 15723.019} C_VEL
LIN {X 0,Y 287.043,Z 966.975,A -85,B 0,C 180,E1 15730.021,E2 15730.021} C_VEL
LIN {X 0,Y 285.585,Z 979.19,A -85,B 0,C 180,E1 15737.383,E2 15737.383} C_VEL
LIN {X 0,Y 285.559,Z 985.471,A -85,B 0,C 180,E1 15743.933,E2 15743.933} C_VEL
LIN {X 0,Y 285.93,Z 987.51,A -85,B 0,C 180,E1 15750,E2 15750} C_VEL
LIN {X 0,Y 285.56,Z 985.48,A -85,B 0,C 180,E1 15756.067,E2 15756.067} C_VEL
LIN {X 0,Y 285.625,Z 979.158,A -85,B 0,C 180,E1 15762.657,E2 15762.657} C_VEL
LIN {X 0,Y 287.033,Z 966.982,A -85,B 0,C 180,E1 15769.985,E2 15769.985} C_VEL
LIN {X 0,Y 291.671,Z 947.784,A -85,B 0,C 180,E1 15777.751,E2 15777.751} C_VEL
LIN {X 0,Y 299.807,Z 922.355,A -85,B 0,C 180,E1 15784.927,E2 15784.927} C_VEL
LIN {X 0,Y 309.951,Z 893.385,A -85,B 0,C 180,E1 15790.761,E2 15790.761} C_VEL
LIN {X 0,Y 321.393,Z 860.34,A -85,B 0,C 180,E1 15795.486,E2 15795.486} C_VEL
LIN {X 0,Y 332.475,Z 824.264,A -85,B 0,C 180,E1 15799.076,E2 15799.076} C_VEL
LIN {X 0,Y 340.403,Z 790.826,A -85,B 0,C 180,E1 15801.434,E2 15801.434} C_VEL
LIN {X 0,Y 337.451,Z 781.346,A -85,B 0,C 180,E1 15802.862,E2 15802.862} C_VEL
LIN {X 0,Y 332.482,Z 773.888,A -85,B 0,C 180,E1 15804.51,E2 15804.51} C_VEL
LIN {X 0,Y 324.151,Z 764.25,A -85,B 0,C 180,E1 15807.186,E2 15807.186} C_VEL
LIN {X 0,Y 323.52,Z 762.799,A -85,B 0,C 180,E1 15807.459,E2 15807.459} C_VEL
LIN {X 0,Y 312.105,Z 739.762,A -85,B 0,C 180,E1 15812.458,E2 15812.458} C_VEL
LIN {X 0,Y 299.857,Z 719.774,A -85,B 0,C 180,E1 15818.307,E2 15818.307} C_VEL
LIN {X 0,Y 290.532,Z 706.526,A -85,B 0,C 180,E1 15823.785,E2 15823.785} C_VEL
LIN {X 0,Y 285.986,Z 699.877,A -85,B 0,C 180,E1 15827.23,E2 15827.23} C_VEL
LIN {X 0,Y 281.908,Z 694.739,A -85,B 0,C 180,E1 15831.127,E2 15831.127} C_VEL
LIN {X 0,Y 281.046,Z 692.652,A -85,B 0,C 180,E1 15832.281,E2 15832.281} C_VEL
LIN {X 0,Y 276.753,Z 688.78,A -85,B 0,C 180,E1 15841.556,E2 15841.556} C_VEL
LIN {X 0,Y 281.149,Z 693.478,A -85,B 0,C 180,E1 15853.97,E2 15853.97} C_VEL
LIN {X 0,Y 283.925,Z 698.874,A -85,B 0,C 180,E1 15857.332,E2 15857.332} C_VEL
LIN {X 0,Y 286.319,Z 701.338,A -85,B 0,C 180,E1 15859.491,E2 15859.491} C_VEL
LIN {X 0,Y 290.008,Z 706.926,A -85,B 0,C 180,E1 15862.558,E2 15862.558} C_VEL
LIN {X 0,Y 298.586,Z 721.84,A -85,B 0,C 180,E1 15868.776,E2 15868.776} C_VEL
LIN {X 0,Y 307.898,Z 740.794,A -85,B 0,C 180,E1 15874.915,E2 15874.915} C_VEL
LIN {X 0,Y 315.561,Z 762.163,A -85,B 0,C 180,E1 15880.546,E2 15880.546} C_VEL
LIN {X 0,Y 320.655,Z 787.663,A -85,B 0,C 180,E1 15886.482,E2 15886.482} C_VEL
LIN {X 0,Y 321.087,Z 798.523,A -85,B 0,C 180,E1 15888.856,E2 15888.856} C_VEL
LIN {X 0,Y 310.086,Z 825.629,A -85,B 0,C 180,E1 15893.424,E2 15893.424} C_VEL
LIN {X 0,Y 299.476,Z 848.491,A -85,B 0,C 180,E1 15898.918,E2 15898.918} C_VEL
LIN {X 0,Y 290.359,Z 867.05,A -85,B 0,C 180,E1 15905.433,E2 15905.433} C_VEL
LIN {X 0,Y 283.717,Z 880.832,A -85,B 0,C 180,E1 15912.873,E2 15912.873} C_VEL
LIN {X 0,Y 280.131,Z 889.095,A -85,B 0,C 180,E1 15920.7,E2 15920.7} C_VEL
LIN {X 0,Y 279.239,Z 891.995,A -85,B 0,C 180,E1 15926.902,E2 15926.902} C_VEL
LIN {X 0,Y 279.239,Z 891.962,A -85,B 0,C 180,E1 15933.098,E2 15933.098} C_VEL
LIN {X 0,Y 280.672,Z 887.768,A -85,B 0,C 180,E1 15940.846,E2 15940.846} C_VEL
LIN {X 0,Y 284.768,Z 878.478,A -85,B 0,C 180,E1 15948.538,E2 15948.538} C_VEL
LIN {X 0,Y 292.226,Z 863.25,A -85,B 0,C 180,E1 15956.035,E2 15956.035} C_VEL
LIN {X 0,Y 302.243,Z 842.645,A -85,B 0,C 180,E1 15962.576,E2 15962.576} C_VEL
LIN {X 0,Y 313.283,Z 817.954,A -85,B 0,C 180,E1 15967.934,E2 15967.934} C_VEL
LIN {X 0,Y 321.531,Z 795.486,A -85,B 0,C 180,E1 15971.583,E2 15971.583} C_VEL
LIN {X 0,Y 317.738,Z 771.133,A -85,B 0,C 180,E1 15977.206,E2 15977.206} C_VEL
LIN {X 0,Y 311.264,Z 749.311,A -85,B 0,C 180,E1 15982.591,E2 15982.591} C_VEL
LIN {X 0,Y 302.536,Z 729.469,A -85,B 0,C 180,E1 15988.425,E2 15988.425} C_VEL
LIN {X 0,Y 293.738,Z 713.168,A -85,B 0,C 180,E1 15994.423,E2 15994.423} C_VEL
LIN {X 0,Y 289.09,Z 706.194,A -85,B 0,C 180,E1 15997.872,E2 15997.872} C_VEL
LIN {X 0,Y 285.174,Z 699.769,A -85,B 0,C 180,E1 16001.296,E2 16001.296} C_VEL
LIN {X 0,Y 281.483,Z 694.795,A -85,B 0,C 180,E1 16005.156,E2 16005.156} C_VEL
LIN {X 0,Y 280.944,Z 692.696,A -85,B 0,C 180,E1 16006.02,E2 16006.02} C_VEL
LIN {X 0,Y 276.445,Z 688.418,A -85,B 0,C 180,E1 16016.877,E2 16016.877} C_VEL
LIN {X 0,Y 277.614,Z 690.102,A -85,B 0,C 180,E1 16022.732,E2 16022.732} C_VEL
LIN {X 0,Y 281.611,Z 693.658,A -85,B 0,C 180,E1 16028.678,E2 16028.678} C_VEL
LIN {X 0,Y 284.635,Z 698.995,A -85,B 0,C 180,E1 16031.86,E2 16031.86} C_VEL
LIN {X 0,Y 287.079,Z 701.442,A -85,B 0,C 180,E1 16033.812,E2 16033.812} C_VEL
LIN {X 0,Y 292.917,Z 710.21,A -85,B 0,C 180,E1 16037.912,E2 16037.912} C_VEL
LIN {X 0,Y 298.294,Z 717.878,A -85,B 0,C 180,E1 16040.988,E2 16040.988} C_VEL
LIN {X 0,Y 308.528,Z 733.899,A -85,B 0,C 180,E1 16046.022,E2 16046.022} C_VEL
LIN {X 0,Y 321.086,Z 757.512,A -85,B 0,C 180,E1 16051.527,E2 16051.527} C_VEL
LIN {X 0,Y 331.97,Z 785.86,A -85,B 0,C 180,E1 16056.539,E2 16056.539} C_VEL
LIN {X 0,Y 334.38,Z 795.657,A -85,B 0,C 180,E1 16057.972,E2 16057.972} C_VEL
LIN {X 0,Y 323.639,Z 834.233,A -85,B 0,C 180,E1 16060.859,E2 16060.859} C_VEL
LIN {X 0,Y 311.975,Z 869.105,A -85,B 0,C 180,E1 16064.761,E2 16064.761} C_VEL
LIN {X 0,Y 300.559,Z 900.219,A -85,B 0,C 180,E1 16069.729,E2 16069.729} C_VEL
LIN {X 0,Y 290.459,Z 927.851,A -85,B 0,C 180,E1 16075.914,E2 16075.914} C_VEL
LIN {X 0,Y 283.058,Z 950.711,A -85,B 0,C 180,E1 16083.055,E2 16083.055} C_VEL
LIN {X 0,Y 278.789,Z 968.661,A -85,B 0,C 180,E1 16091.049,E2 16091.049} C_VEL
LIN {X 0,Y 277.751,Z 978.924,A -85,B 0,C 180,E1 16097.946,E2 16097.946} C_VEL
LIN {X 0,Y 277.731,Z 984.144,A -85,B 0,C 180,E1 16103.762,E2 16103.762} C_VEL
LIN {X 0,Y 278.141,Z 986.198,A -85,B 0,C 180,E1 16110,E2 16110} C_VEL
LIN {X 0,Y 277.73,Z 984.153,A -85,B 0,C 180,E1 16116.238,E2 16116.238} C_VEL
LIN {X 0,Y 277.8,Z 977.41,A -85,B 0,C 180,E1 16123.348,E2 16123.348} C_VEL
LIN {X 0,Y 279.667,Z 964.027,A -85,B 0,C 180,E1 16131.359,E2 16131.359} C_VEL
LIN {X 0,Y 284.776,Z 944.904,A -85,B 0,C 180,E1 16139.023,E2 16139.023} C_VEL
LIN {X 0,Y 293.019,Z 920.902,A -85,B 0,C 180,E1 16145.859,E2 16145.859} C_VEL
LIN {X 0,Y 303.842,Z 891.56,A -85,B 0,C 180,E1 16151.841,E2 16151.841} C_VEL
LIN {X 0,Y 315.655,Z 858.802,A -85,B 0,C 180,E1 16156.555,E2 16156.555} C_VEL
LIN {X 0,Y 327.326,Z 822.163,A -85,B 0,C 180,E1 16160.197,E2 16160.197} C_VEL
LIN {X 0,Y 334.549,Z 794.203,A -85,B 0,C 180,E1 16162.166,E2 16162.166} C_VEL
LIN {X 0,Y 324.465,Z 764.853,A -85,B 0,C 180,E1 16167.061,E2 16167.061} C_VEL
LIN {X 0,Y 323.52,Z 762.799,A -85,B 0,C 180,E1 16167.459,E2 16167.459} C_VEL
LIN {X 0,Y 319.732,Z 759.081,A -85,B 0,C 180,E1 16168.711,E2 16168.711} C_VEL
LIN {X 0,Y 313.298,Z 755.342,A -85,B 0,C 180,E1 16170.757,E2 16170.757} C_VEL
LIN {X 0,Y 312.851,Z 754.483,A -85,B 0,C 180,E1 16170.964,E2 16170.964} C_VEL
LIN {X 0,Y 300.831,Z 732.66,A -85,B 0,C 180,E1 16176.855,E2 16176.855} C_VEL
LIN {X 0,Y 292.276,Z 719.48,A -85,B 0,C 180,E1 16181.755,E2 16181.755} C_VEL
LIN {X 0,Y 288.023,Z 713.359,A -85,B 0,C 180,E1 16184.615,E2 16184.615} C_VEL
LIN {X 0,Y 284.038,Z 707.27,A -85,B 0,C 180,E1 16187.869,E2 16187.869} C_VEL
LIN {X 0,Y 280.277,Z 701.603,A -85,B 0,C 180,E1 16191.855,E2 16191.855} C_VEL
LIN {X 0,Y 278.539,Z 699.814,A -85,B 0,C 180,E1 16194.164,E2 16194.164} C_VEL
LIN {X 0,Y 275.728,Z 696.612,A -85,B 0,C 180,E1 16201.562,E2 16201.562} C_VEL
LIN {X 0,Y 279.571,Z 701.228,A -85,B 0,C 180,E1 16213.632,E2 16213.632} C_VEL
LIN {X 0,Y 282.54,Z 706.822,A -85,B 0,C 180,E1 16217.475,E2 16217.475} C_VEL
LIN {X 0,Y 284.241,Z 709.082,A -85,B 0,C 180,E1 16219.169,E2 16219.169} C_VEL
LIN {X 0,Y 288.911,Z 717.446,A -85,B 0,C 180,E1 16223.461,E2 16223.461} C_VEL
LIN {X 0,Y 294.845,Z 727.641,A -85,B 0,C 180,E1 16228.008,E2 16228.008} C_VEL
LIN {X 0,Y 303.535,Z 746.843,A -85,B 0,C 180,E1 16234.427,E2 16234.427} C_VEL
LIN {X 0,Y 310.438,Z 768.112,A -85,B 0,C 180,E1 16240.236,E2 16240.236} C_VEL
LIN {X 0,Y 314.564,Z 791.949,A -85,B 0,C 180,E1 16246.007,E2 16246.007} C_VEL
LIN {X 0,Y 315.227,Z 799.945,A -85,B 0,C 180,E1 16247.919,E2 16247.919} C_VEL
LIN {X 0,Y 303.615,Z 827.539,A -85,B 0,C 180,E1 16252.661,E2 16252.661} C_VEL
LIN {X 0,Y 292.811,Z 849.835,A -85,B 0,C 180,E1 16258.129,E2 16258.129} C_VEL
LIN {X 0,Y 282.978,Z 868.929,A -85,B 0,C 180,E1 16265.007,E2 16265.007} C_VEL
LIN {X 0,Y 275.817,Z 882.927,A -85,B 0,C 180,E1 16272.99,E2 16272.99} C_VEL
LIN {X 0,Y 272.452,Z 890.405,A -85,B 0,C 180,E1 16280.436,E2 16280.436} C_VEL
LIN {X 0,Y 271.474,Z 893.304,A -85,B 0,C 180,E1 16286.814,E2 16286.814} C_VEL
LIN {X 0,Y 271.474,Z 893.272,A -85,B 0,C 180,E1 16293.186,E2 16293.186} C_VEL
LIN {X 0,Y 273.001,Z 889.086,A -85,B 0,C 180,E1 16301.155,E2 16301.155} C_VEL
LIN {X 0,Y 277.369,Z 879.801,A -85,B 0,C 180,E1 16309.052,E2 16309.052} C_VEL
LIN {X 0,Y 285.223,Z 864.581,A -85,B 0,C 180,E1 16316.724,E2 16316.724} C_VEL
LIN {X 0,Y 294.998,Z 845.49,A -85,B 0,C 180,E1 16322.998,E2 16322.998} C_VEL
LIN {X 0,Y 306.487,Z 820.922,A -85,B 0,C 180,E1 16328.535,E2 16328.535} C_VEL
LIN {X 0,Y 315.258,Z 799.396,A -85,B 0,C 180,E1 16332.076,E2 16332.076} C_VEL
LIN {X 0,Y 311.906,Z 774.828,A -85,B 0,C 180,E1 16337.979,E2 16337.979} C_VEL
LIN {X 0,Y 305.799,Z 752.814,A -85,B 0,C 180,E1 16343.7,E2 16343.7} C_VEL
LIN {X 0,Y 297.238,Z 732.35,A -85,B 0,C 180,E1 16350.062,E2 16350.062} C_VEL
LIN {X 0,Y 289.793,Z 718.954,A -85,B 0,C 180,E1 16355.595,E2 16355.595} C_VEL
LIN {X 0,Y 286.371,Z 713.211,A -85,B 0,C 180,E1 16358.464,E2 16358.464} C_VEL
LIN {X 0,Y 283.1,Z 707.171,A -85,B 0,C 180,E1 16361.758,E2 16361.758} C_VEL
LIN {X 0,Y 279.669,Z 701.899,A -85,B 0,C 180,E1 16365.756,E2 16365.756} C_VEL
LIN {X 0,Y 278.863,Z 700.23,A -85,B 0,C 180,E1 16367.051,E2 16367.051} C_VEL
LIN {X 0,Y 275.498,Z 696.32,A -85,B 0,C 180,E1 16378.437,E2 16378.437} C_VEL
LIN {X 0,Y 280.209,Z 701.458,A -85,B 0,C 180,E1 16388.299,E2 16388.299} C_VEL
LIN {X 0,Y 283.784,Z 707.097,A -85,B 0,C 180,E1 16392.091,E2 16392.091} C_VEL
LIN {X 0,Y 285.856,Z 710.274,A -85,B 0,C 180,E1 16393.873,E2 16393.873} C_VEL
LIN {X 0,Y 290.874,Z 717.504,A -85,B 0,C 180,E1 16397.457,E2 16397.457} C_VEL
LIN {X 0,Y 298.404,Z 728.832,A -85,B 0,C 180,E1 16401.944,E2 16401.944} C_VEL
LIN {X 0,Y 310.371,Z 749.896,A -85,B 0,C 180,E1 16407.939,E2 16407.939} C_VEL
LIN {X 0,Y 320.974,Z 773.798,A -85,B 0,C 180,E1 16413.014,E2 16413.014} C_VEL
LIN {X 0,Y 328.478,Z 797.042,A -85,B 0,C 180,E1 16417.024,E2 16417.024} C_VEL
LIN {X 0,Y 317.865,Z 834.047,A -85,B 0,C 180,E1 16419.876,E2 16419.876} C_VEL
LIN {X 0,Y 305.9,Z 868.398,A -85,B 0,C 180,E1 16423.773,E2 16423.773} C_VEL
LIN {X 0,Y 294.28,Z 898.747,A -85,B 0,C 180,E1 16428.685,E2 16428.685} C_VEL
LIN {X 0,Y 283.563,Z 926.394,A -85,B 0,C 180,E1 16434.965,E2 16434.965} C_VEL
LIN {X 0,Y 275.644,Z 949.282,A -85,B 0,C 180,E1 16442.269,E2 16442.269} C_VEL
LIN {X 0,Y 271.075,Z 967.273,A -85,B 0,C 180,E1 16450.488,E2 16450.488} C_VEL
LIN {X 0,Y 269.917,Z 977.981,A -85,B 0,C 180,E1 16457.95,E2 16457.95} C_VEL
LIN {X 0,Y 269.923,Z 982.82,A -85,B 0,C 180,E1 16463.58,E2 16463.58} C_VEL
LIN {X 0,Y 270.348,Z 984.887,A -85,B 0,C 180,E1 16470,E2 16470} C_VEL
LIN {X 0,Y 269.921,Z 982.829,A -85,B 0,C 180,E1 16476.42,E2 16476.42} C_VEL
LIN {X 0,Y 269.971,Z 976.05,A -85,B 0,C 180,E1 16483.742,E2 16483.742} C_VEL
LIN {X 0,Y 272.034,Z 962.631,A -85,B 0,C 180,E1 16491.989,E2 16491.989} C_VEL
LIN {X 0,Y 277.644,Z 943.019,A -85,B 0,C 180,E1 16500.01,E2 16500.01} C_VEL
LIN {X 0,Y 286.736,Z 918.461,A -85,B 0,C 180,E1 16507.069,E2 16507.069} C_VEL
LIN {X 0,Y 297.728,Z 890.083,A -85,B 0,C 180,E1 16512.904,E2 16512.904} C_VEL
LIN {X 0,Y 310.062,Z 857.277,A -85,B 0,C 180,E1 16517.658,E2 16517.658} C_VEL
LIN {X 0,Y 322.106,Z 820.702,A -85,B 0,C 180,E1 16521.3,E2 16521.3} C_VEL
LIN {X 0,Y 328.432,Z 796.546,A -85,B 0,C 180,E1 16523.069,E2 16523.069} C_VEL
LIN {X 0,Y 318.873,Z 768.074,A -85,B 0,C 180,E1 16528.1,E2 16528.1} C_VEL
LIN {X 0,Y 312.851,Z 754.483,A -85,B 0,C 180,E1 16530.964,E2 16530.964} C_VEL
LIN {X 0,Y 309.315,Z 751.271,A -85,B 0,C 180,E1 16532.313,E2 16532.313} C_VEL
LIN {X 0,Y 302.557,Z 748.151,A -85,B 0,C 180,E1 16534.762,E2 16534.762} C_VEL
LIN {X 0,Y 291.234,Z 728.188,A -85,B 0,C 180,E1 16541.37,E2 16541.37} C_VEL
LIN {X 0,Y 282.395,Z 714.808,A -85,B 0,C 180,E1 16548.224,E2 16548.224} C_VEL
LIN {X 0,Y 278.69,Z 708.964,A -85,B 0,C 180,E1 16552.363,E2 16552.363} C_VEL
LIN {X 0,Y 274.589,Z 704.407,A -85,B 0,C 180,E1 16561.568,E2 16561.568} C_VEL
LIN {X 0,Y 277.801,Z 709.047,A -85,B 0,C 180,E1 16573.341,E2 16573.341} C_VEL
LIN {X 0,Y 280.84,Z 714.608,A -85,B 0,C 180,E1 16577.585,E2 16577.585} C_VEL
LIN {X 0,Y 286.08,Z 724.574,A -85,B 0,C 180,E1 16583.075,E2 16583.075} C_VEL
LIN {X 0,Y 292.091,Z 736.097,A -85,B 0,C 180,E1 16588.159,E2 16588.159} C_VEL
LIN {X 0,Y 300.018,Z 755.19,A -85,B 0,C 180,E1 16594.663,E2 16594.663} C_VEL
LIN {X 0,Y 305.571,Z 775.52,A -85,B 0,C 180,E1 16600.306,E2 16600.306} C_VEL
LIN {X 0,Y 308.789,Z 799.315,A -85,B 0,C 180,E1 16606.291,E2 16606.291} C_VEL
LIN {X 0,Y 308.206,Z 804.662,A -85,B 0,C 180,E1 16607.457,E2 16607.457} C_VEL
LIN {X 0,Y 296.206,Z 831.582,A -85,B 0,C 180,E1 16612.314,E2 16612.314} C_VEL
LIN {X 0,Y 284.374,Z 854.732,A -85,B 0,C 180,E1 16618.399,E2 16618.399} C_VEL
LIN {X 0,Y 274.658,Z 872.506,A -85,B 0,C 180,E1 16625.405,E2 16625.405} C_VEL
LIN {X 0,Y 267.834,Z 885.204,A -85,B 0,C 180,E1 16633.258,E2 16633.258} C_VEL
LIN {X 0,Y 264.757,Z 891.72,A -85,B 0,C 180,E1 16640.155,E2 16640.155} C_VEL
LIN {X 0,Y 263.713,Z 894.613,A -85,B 0,C 180,E1 16646.72,E2 16646.72} C_VEL
LIN {X 0,Y 263.713,Z 894.581,A -85,B 0,C 180,E1 16653.28,E2 16653.28} C_VEL
LIN {X 0,Y 265.336,Z 890.404,A -85,B 0,C 180,E1 16661.481,E2 16661.481} C_VEL
LIN {X 0,Y 269.978,Z 881.125,A -85,B 0,C 180,E1 16669.594,E2 16669.594} C_VEL
LIN {X 0,Y 278.258,Z 865.914,A -85,B 0,C 180,E1 16677.449,E2 16677.449} C_VEL
LIN {X 0,Y 289.029,Z 845.728,A -85,B 0,C 180,E1 16684.141,E2 16684.141} C_VEL
LIN {X 0,Y 300.269,Z 822.714,A -85,B 0,C 180,E1 16689.38,E2 16689.38} C_VEL
LIN {X 0,Y 308.884,Z 802.047,A -85,B 0,C 180,E1 16692.891,E2 16692.891} C_VEL
LIN {X 0,Y 306.177,Z 778.901,A -85,B 0,C 180,E1 16698.694,E2 16698.694} C_VEL
LIN {X 0,Y 301.093,Z 758.675,A -85,B 0,C 180,E1 16704.157,E2 16704.157} C_VEL
LIN {X 0,Y 293.243,Z 738.381,A -85,B 0,C 180,E1 16710.745,E2 16710.745} C_VEL
LIN {X 0,Y 284.719,Z 721.39,A -85,B 0,C 180,E1 16718.106,E2 16718.106} C_VEL
LIN {X 0,Y 280.583,Z 714.354,A -85,B 0,C 180,E1 16722.399,E2 16722.399} C_VEL
LIN {X 0,Y 277.707,Z 708.724,A -85,B 0,C 180,E1 16726.467,E2 16726.467} C_VEL
LIN {X 0,Y 274.256,Z 704.124,A -85,B 0,C 180,E1 16736.852,E2 16736.852} C_VEL
LIN {X 0,Y 275.715,Z 706.233,A -85,B 0,C 180,E1 16743.364,E2 16743.364} C_VEL
LIN {X 0,Y 278.693,Z 709.121,A -85,B 0,C 180,E1 16747.923,E2 16747.923} C_VEL
LIN {X 0,Y 282.401,Z 714.841,A -85,B 0,C 180,E1 16751.955,E2 16751.955} C_VEL
LIN {X 0,Y 288.94,Z 725.38,A -85,B 0,C 180,E1 16757.284,E2 16757.284} C_VEL
LIN {X 0,Y 296.141,Z 736.919,A -85,B 0,C 180,E1 16761.799,E2 16761.799} C_VEL
LIN {X 0,Y 306.544,Z 756.357,A -85,B 0,C 180,E1 16767.437,E2 16767.437} C_VEL
LIN {X 0,Y 316.266,Z 779.339,A -85,B 0,C 180,E1 16772.467,E2 16772.467} C_VEL
LIN {X 0,Y 322.442,Z 799.939,A -85,B 0,C 180,E1 16776.182,E2 16776.182} C_VEL
LIN {X 0,Y 311.28,Z 836.692,A -85,B 0,C 180,E1 16779.138,E2 16779.138} C_VEL
LIN {X 0,Y 298.445,Z 871.531,A -85,B 0,C 180,E1 16783.279,E2 16783.279} C_VEL
LIN {X 0,Y 285.796,Z 902.901,A -85,B 0,C 180,E1 16788.701,E2 16788.701} C_VEL
LIN {X 0,Y 274.757,Z 930.227,A -85,B 0,C 180,E1 16795.473,E2 16795.473} C_VEL
LIN {X 0,Y 267.066,Z 952.014,A -85,B 0,C 180,E1 16803.127,E2 16803.127} C_VEL
LIN {X 0,Y 263.05,Z 967.673,A -85,B 0,C 180,E1 16810.973,E2 16810.973} C_VEL
LIN {X 0,Y 262.073,Z 977.312,A -85,B 0,C 180,E1 16818.204,E2 16818.204} C_VEL
LIN {X 0,Y 262.089,Z 981.492,A -85,B 0,C 180,E1 16823.388,E2 16823.388} C_VEL
LIN {X 0,Y 262.558,Z 983.575,A -85,B 0,C 180,E1 16830,E2 16830} C_VEL
LIN {X 0,Y 262.084,Z 981.501,A -85,B 0,C 180,E1 16836.612,E2 16836.612} C_VEL
LIN {X 0,Y 262.177,Z 974.695,A -85,B 0,C 180,E1 16844.159,E2 16844.159} C_VEL
LIN {X 0,Y 264.425,Z 961.234,A -85,B 0,C 180,E1 16852.656,E2 16852.656} C_VEL
LIN {X 0,Y 270.672,Z 941.141,A -85,B 0,C 180,E1 16861.043,E2 16861.043} C_VEL
LIN {X 0,Y 280.528,Z 916.034,A -85,B 0,C 180,E1 16868.334,E2 16868.334} C_VEL
LIN {X 0,Y 292.433,Z 886.843,A -85,B 0,C 180,E1 16874.319,E2 16874.319} C_VEL
LIN {X 0,Y 305.577,Z 853.097,A -85,B 0,C 180,E1 16879.126,E2 16879.126} C_VEL
LIN {X 0,Y 317.887,Z 816.378,A -85,B 0,C 180,E1 16882.665,E2 16882.665} C_VEL
LIN {X 0,Y 322.436,Z 799.626,A -85,B 0,C 180,E1 16883.887,E2 16883.887} C_VEL
LIN {X 0,Y 313.434,Z 771.408,A -85,B 0,C 180,E1 16889.11,E2 16889.11} C_VEL
LIN {X 0,Y 302.702,Z 748.372,A -85,B 0,C 180,E1 16894.691,E2 16894.691} C_VEL
LIN {X 0,Y 302.557,Z 748.151,A -85,B 0,C 180,E1 16894.762,E2 16894.762} C_VEL
LIN {X 0,Y 295.829,Z 743.175,A -85,B 0,C 180,E1 16897.731,E2 16897.731} C_VEL
LIN {X 0,Y 289.965,Z 738.122,A -85,B 0,C 180,E1 16900.822,E2 16900.822} C_VEL
LIN {X 0,Y 283.327,Z 727.367,A -85,B 0,C 180,E1 16905.833,E2 16905.833} C_VEL
LIN {X 0,Y 280.012,Z 721.955,A -85,B 0,C 180,E1 16908.954,E2 16908.954} C_VEL
LIN {X 0,Y 276.315,Z 715.579,A -85,B 0,C 180,E1 16913.724,E2 16913.724} C_VEL
LIN {X 0,Y 273.168,Z 712.179,A -85,B 0,C 180,E1 16921.577,E2 16921.577} C_VEL
